(* CODESYS project TheWorld
   CompiledLibraryCompatibilityVersion: CODESYS V3.5 SP16 Patch 2

Project tree, tasks and I/O mapping:
  Device : CODESYS Control for Linux SL, CODESYS GmbH, order no. 2302000005, version 4.8.0.0
    application Application
      AC_FBs/
      AC_RMP/
      AC_Std/
      Alarm Configuration
      program BlinkingAlarm [CFC]
      program Calculus [ST]
      visualisation Chiller1Menu
      text list Chiller2Alarmgroup
      program Chiller_1 [ST]
      Chiller_func/
      text list Chiller_trendvalues
      function block ConvertDataArray_1 [ST]
      function block ConvertDataArray_2 [ST]
      function block ConvertDataArray_3 [ST]
      function block ConvertDataArray [ST]
      Enums/
    Ethernet : Ethernet, 3S - Smart Software Solutions GmbH, version 4.1.0.0 (disabled)
        settings: IPAddress = [172,16,0,11]; SubnetMask = [255,255,255,0]; GatewayAddress = [172,16,0,1]; MACAddress = [16#00,16#00,16#00,16#00,16#00,16#00]; NetworkInterfaceName = 'eno1'; NetworkInterfaceName = "eno1"; SaveCommunicationSettings = FALSE; IPAddress = [192,168,0,2]; SubnetMask = [255,255,255,0]; GatewayAddress = [0,0,0,0]
      Modbus_TCP_Master : Modbus TCP Master, 3S - Smart Software Solutions GmbH, version 4.2.0.0
          settings: AutoReconnect = TRUE
        Modbus_TCP_Slave_AC1 : Modbus TCP Slave, 3S - Smart Software Solutions GmbH, version 4.1.0.0
            settings: Unit-ID = 255; IPAddress = [192, 168, 0, 51]; Channel 0.Function Code = 3; Channel 0.Read Offset = 16#0000; Channel 0.Read Length = 124; Channel 0.Write Offset = 0; Channel 0.Write Length = 0; Channel 0.Cycle Time = 100; Channel 1.Function Code = 3; Channel 1.Read Offset = 16#007C; Channel 1.Read Length = 124; Channel 1.Write Offset = 0; Channel 1.Write Length = 0; Channel 1.Cycle Time = 100; Channel 2.Function Code = 3; Channel 2.Read Offset = 16#00F8; Channel 2.Read Length = 124; Channel 2.Write Offset = 0; Channel 2.Write Length = 0; Channel 2.Cycle Time = 100; Channel 3.Function Code = 16; Channel 3.Read Offset = 0; Channel 3.Read Length = 0; Channel 3.Write Offset = 16#011E; Channel 3.Write Length = 4; Channel 3.Cycle Time = 100
            input  Application.Chiller_1.modbus_var_1000 : ARRAY[0..123] OF WORD  // Channel 0
            input  Application.Chiller_1.modbus_var_1001 : ARRAY[0..123] OF WORD  // Channel 1
            input  Application.Chiller_1.modbus_var_1002 : ARRAY[0..123] OF WORD  // Channel 2
            output Application.Chiller_1.modbus_var_1002[286] : WORD  // Channel 3.Channel 3
            output Application.Chiller_1.modbus_var_1002[287] : WORD  // Channel 3.Channel 3
            output Application.Chiller_1.modbus_var_1002[288] : WORD  // Channel 3.Channel 3
            output Application.Chiller_1.modbus_var_1002[289] : WORD  // Channel 3.Channel 3
            unmapped channels: Channel 3
        Modbus_TCP_Slave_AC2 : Modbus TCP Slave, 3S - Smart Software Solutions GmbH, version 4.1.0.0
            settings: Unit-ID = 255; IPAddress = [192, 168, 0, 52]; Channel 0.Function Code = 3; Channel 0.Read Offset = 16#0000; Channel 0.Read Length = 124; Channel 0.Write Offset = 0; Channel 0.Write Length = 0; Channel 0.Cycle Time = 100; Channel 1.Function Code = 3; Channel 1.Read Offset = 16#007C; Channel 1.Read Length = 124; Channel 1.Write Offset = 0; Channel 1.Write Length = 0; Channel 1.Cycle Time = 100; Channel 2.Function Code = 3; Channel 2.Read Offset = 16#012C; Channel 2.Read Length = 100; Channel 2.Write Offset = 0; Channel 2.Write Length = 0; Channel 2.Cycle Time = 100
            input  Application.Chiller_2.modbus_var_1000 : ARRAY[0..123] OF WORD  // Channel 0
            input  Application.Chiller_2.modbus_var_1001 : ARRAY[0..123] OF WORD  // Channel 1
            input  Application.Chiller_2.modbus_var_1002 : ARRAY[0..99] OF WORD  // Channel 2
        Modbus_TCP_Slave_AC3 : Modbus TCP Slave, 3S - Smart Software Solutions GmbH, version 4.1.0.0
            settings: Unit-ID = 255; IPAddress = [192, 168, 0, 53]; Channel 0.Function Code = 3; Channel 0.Read Offset = 16#0000; Channel 0.Read Length = 124; Channel 0.Write Offset = 0; Channel 0.Write Length = 0; Channel 0.Cycle Time = 100; Channel 1.Function Code = 3; Channel 1.Read Offset = 16#007C; Channel 1.Read Length = 124; Channel 1.Write Offset = 0; Channel 1.Write Length = 0; Channel 1.Cycle Time = 100; Channel 2.Function Code = 3; Channel 2.Read Offset = 16#00F8; Channel 2.Read Length = 124; Channel 2.Write Offset = 0; Channel 2.Write Length = 0; Channel 2.Cycle Time = 100; Channel 3.Function Code = 16; Channel 3.Read Offset = 0; Channel 3.Read Length = 0; Channel 3.Write Offset = 16#011E; Channel 3.Write Length = 4; Channel 3.Cycle Time = 100
            input  Application.Chiller_3.modbus_var_1000 : ARRAY[0..123] OF WORD  // Channel 0
            input  Application.Chiller_3.modbus_var_1001 : ARRAY[0..123] OF WORD  // Channel 1
            input  Application.Chiller_3.modbus_var_1002 : ARRAY[0..123] OF WORD  // Channel 2
            output Application.Chiller_3.modbus_var_1002[286] : WORD  // Channel 3.Channel 3
            output Application.Chiller_3.modbus_var_1002[287] : WORD  // Channel 3.Channel 3
            output Application.Chiller_3.modbus_var_1002[288] : WORD  // Channel 3.Channel 3
            output Application.Chiller_3.modbus_var_1002[289] : WORD  // Channel 3.Channel 3
            unmapped channels: Channel 3
        Modbus_TCP_Slave_AC4 : Modbus TCP Slave, 3S - Smart Software Solutions GmbH, version 4.1.0.0
            settings: Unit-ID = 255; IPAddress = [192, 168, 0, 54]; Channel 0.Function Code = 3; Channel 0.Read Offset = 16#0000; Channel 0.Read Length = 124; Channel 0.Write Offset = 0; Channel 0.Write Length = 0; Channel 0.Cycle Time = 100; Channel 1.Function Code = 3; Channel 1.Read Offset = 16#007C; Channel 1.Read Length = 124; Channel 1.Write Offset = 0; Channel 1.Write Length = 0; Channel 1.Cycle Time = 100; Channel 2.Function Code = 3; Channel 2.Read Offset = 16#012C; Channel 2.Read Length = 100; Channel 2.Write Offset = 0; Channel 2.Write Length = 0; Channel 2.Cycle Time = 100
            input  Application.Chiller_4.modbus_var_1000 : ARRAY[0..123] OF WORD  // Channel 0
            input  Application.Chiller_4.modbus_var_1001 : ARRAY[0..123] OF WORD  // Channel 1
            input  Application.Chiller_4.modbus_var_1002 : ARRAY[0..99] OF WORD  // Channel 2
    Modbus_COM_1 : Modbus COM, 3S - Smart Software Solutions GmbH, version 3.5.16.0
        settings: DataBits = 8; StopBits = 1; ComPort = 1
      Modbus_Master_COM_Port_1 : Modbus Master, COM Port, 3S - Smart Software Solutions GmbH, version 4.2.0.0
          settings: Auto-restart communication = TRUE
        Modbus_Slave_COM_Port_AC1 : Modbus Slave, COM Port, 3S - Smart Software Solutions GmbH, version 3.5.16.0
            settings: SlaveAddress = 15; ResponseTimeout = 1000; UseExtendedFunctionCodes = TRUE; Channel 0.Function Code = 3; Channel 0.Read Offset = 16#0000; Channel 0.Read Length = 100; Channel 0.Write Offset = 0; Channel 0.Write Length = 0; Channel 0.Cycle Time = 100
            input  Application.Chiller_1.modbus_var_1000 : ARRAY[0..99] OF WORD  // Channel 0
        Modbus_Slave_COM_Port_AC2 : Modbus Slave, COM Port, 3S - Smart Software Solutions GmbH, version 3.5.16.0
            settings: SlaveAddress = 15; ResponseTimeout = 1000; UseExtendedFunctionCodes = TRUE; Channel 0.Function Code = 3; Channel 0.Read Offset = 16#0200; Channel 0.Read Length = 100; Channel 0.Write Offset = 0; Channel 0.Write Length = 0; Channel 0.Cycle Time = 100
            input  Application.Chiller_2.modbus_var_1000 : ARRAY[0..99] OF WORD  // Channel 0
        Modbus_Slave_COM_Port_AC3 : Modbus Slave, COM Port, 3S - Smart Software Solutions GmbH, version 3.5.16.0
            settings: SlaveAddress = 16; ResponseTimeout = 1000; UseExtendedFunctionCodes = TRUE; Channel 0.Function Code = 3; Channel 0.Read Offset = 16#0400; Channel 0.Read Length = 100; Channel 0.Write Offset = 0; Channel 0.Write Length = 0; Channel 0.Cycle Time = 100
            input  Application.Chiller_3.modbus_var_1000 : ARRAY[0..99] OF WORD  // Channel 0
        Modbus_Slave_COM_Port_AC4 : Modbus Slave, COM Port, 3S - Smart Software Solutions GmbH, version 3.5.16.0
            settings: SlaveAddress = 16; ResponseTimeout = 1000; UseExtendedFunctionCodes = TRUE; Channel 0.Function Code = 3; Channel 0.Read Offset = 16#0600; Channel 0.Read Length = 100; Channel 0.Write Offset = 0; Channel 0.Write Length = 0; Channel 0.Cycle Time = 100
            input  Application.Chiller_4.modbus_var_1000 : ARRAY[0..99] OF WORD  // Channel 0
        Modbus_Slave_COM_Port_AC5 : Modbus Slave, COM Port, 3S - Smart Software Solutions GmbH, version 3.5.16.0
            settings: SlaveAddress = 16; ResponseTimeout = 1000; UseExtendedFunctionCodes = TRUE; Channel 0.Function Code = 3; Channel 0.Read Offset = 16#0800; Channel 0.Read Length = 100; Channel 0.Write Offset = 0; Channel 0.Write Length = 0; Channel 0.Cycle Time = 100
            input  Application.Chiller_5.modbus_var_1000 : ARRAY[0..99] OF WORD  // Channel 0
        Modbus_Slave_COM_Port_AC6 : Modbus Slave, COM Port, 3S - Smart Software Solutions GmbH, version 3.5.16.0
            settings: SlaveAddress = 16; ResponseTimeout = 1000; UseExtendedFunctionCodes = TRUE; Channel 0.Function Code = 3; Channel 0.Read Offset = 16#0C00; Channel 0.Read Length = 100; Channel 0.Write Offset = 0; Channel 0.Write Length = 0; Channel 0.Cycle Time = 100
            input  Application.Chiller_6.modbus_var_1000 : ARRAY[0..99] OF WORD  // Channel 0
        Modbus_Slave_COM_Seq : Modbus Slave, COM Port, 3S - Smart Software Solutions GmbH, version 3.5.16.0
            settings: SlaveAddress = 16; ResponseTimeout = 1000; UseExtendedFunctionCodes = TRUE; Channel 0.Function Code = 3; Channel 0.Read Offset = 16#0A00; Channel 0.Read Length = 108; Channel 0.Write Offset = 0; Channel 0.Write Length = 0; Channel 0.Cycle Time = 100; Channel 1.Function Code = 3; Channel 1.Read Offset = 16#0A7C; Channel 1.Read Length = 83; Channel 1.Write Offset = 0; Channel 1.Write Length = 0; Channel 1.Cycle Time = 100
            input  Application.Sequence.modbus_var_1000 : ARRAY[0..107] OF WORD  // Channel 0
            input  Application.Sequence.modbus_var_add : ARRAY[0..82] OF WORD  // Channel 1
    Modbus_COM_1 : Modbus COM, 3S - Smart Software Solutions GmbH, version 4.1.0.0
      Modbus_Master_COM_Port_1 : Modbus Master, COM Port, 3S - Smart Software Solutions GmbH, version 4.3.0.0
          settings: Transmission = 'RTU'; ResponseTimeout = 1000; TimeBetweenFrames = 10; Auto-restart communication = TRUE
        Modbus_Slave_AC1 : Modbus Slave, COM Port, 3S - Smart Software Solutions GmbH, version 4.1.0.0
            settings: SlaveAddress = 15; ResponseTimeout = 1000; UseExtendedFunctionCodes = TRUE; Channel 0.Function Code = 3; Channel 0.Read Offset = 16#0000; Channel 0.Read Length = 60; Channel 0.Write Offset = 0; Channel 0.Write Length = 0; Channel 0.Cycle Time = 100
            input  Application.Chiller_1.modbus_var_1000 : ARRAY[0..59] OF WORD  // Channel 0
        Modbus_Slave_AC2 : Modbus Slave, COM Port, 3S - Smart Software Solutions GmbH, version 4.1.0.0
            settings: SlaveAddress = 15; ResponseTimeout = 1000; UseExtendedFunctionCodes = TRUE; Channel 0.Function Code = 3; Channel 0.Read Offset = 16#0200; Channel 0.Read Length = 60; Channel 0.Write Offset = 0; Channel 0.Write Length = 0; Channel 0.Cycle Time = 100
            input  Application.Chiller_2.modbus_var_1000 : ARRAY[0..59] OF WORD  // Channel 0
        Modbus_Slave_AC3 : Modbus Slave, COM Port, 3S - Smart Software Solutions GmbH, version 4.1.0.0
            settings: SlaveAddress = 15; ResponseTimeout = 1000; UseExtendedFunctionCodes = TRUE; Channel 0.Function Code = 3; Channel 0.Read Offset = 16#0400; Channel 0.Read Length = 60; Channel 0.Write Offset = 0; Channel 0.Write Length = 0; Channel 0.Cycle Time = 100
            input  Application.Chiller_3.modbus_var_1000 : ARRAY[0..59] OF WORD  // Channel 0
    SoftMotion General Axis Pool
  libraries: CmpBitmapPool, 3.5.17.0 (System); AC_DataLog, 3.5.16.0 (3S - Smart Software Solutions GmbH)
  5ce3da45-db07-42e7-a21c-a00fff4ed8f6|C:\Users\Codesys\Desktop\FlowDiagram_Edited.PNG
  5ce3da45-db07-42e7-a21c-a00fff4ed8f6|C:\Users\Codesys\Desktop\FlowDiagram_Edited.PNG
  5ce3da45-db07-42e7-a21c-a00fff4ed8f6|C:\Users\Codesys\Desktop\Images\Assets från KT_PC\VSD\VSD.jpg
  5ce3da45-db07-42e7-a21c-a00fff4ed8f6|C:\Users\Codesys\Desktop\Images\Assets från KT_PC\VSD\VSD.jpg
  5ce3da45-db07-42e7-a21c-a00fff4ed8f6|C:\Users\Codesys\Desktop\Images\Div bilder\Arrow gray left.png
  5ce3da45-db07-42e7-a21c-a00fff4ed8f6|C:\Users\Codesys\Desktop\Images\Div bilder\Arrow gray left.png
  5ce3da45-db07-42e7-a21c-a00fff4ed8f6|C:\Users\Codesys\Desktop\Images\Div bilder\Arrow green down.png
  5ce3da45-db07-42e7-a21c-a00fff4ed8f6|C:\Users\Codesys\Desktop\Images\Div bilder\Arrow green down.png
  5ce3da45-db07-42e7-a21c-a00fff4ed8f6|C:\Users\Codesys\Desktop\Images\Div bilder\Arrow green up.png
  5ce3da45-db07-42e7-a21c-a00fff4ed8f6|C:\Users\Codesys\Desktop\Images\Div bilder\Arrow green up.png
  5ce3da45-db07-42e7-a21c-a00fff4ed8f6|C:\Users\Codesys\Desktop\Images\Div bilder\Arrow lightblue left.png
  5ce3da45-db07-42e7-a21c-a00fff4ed8f6|C:\Users\Codesys\Desktop\Images\Div bilder\Arrow lightblue left.png
  5ce3da45-db07-42e7-a21c-a00fff4ed8f6|C:\Users\Codesys\Desktop\Images\Div bilder\Arrow red down.png
  5ce3da45-db07-42e7-a21c-a00fff4ed8f6|C:\Users\Codesys\Desktop\Images\Div bilder\Arrow red down.png
  5ce3da45-db07-42e7-a21c-a00fff4ed8f6|C:\Users\Codesys\Desktop\Images\Div bilder\Arrow red left.png
  5ce3da45-db07-42e7-a21c-a00fff4ed8f6|C:\Users\Codesys\Desktop\Images\Div bilder\Arrow red left.png
  5ce3da45-db07-42e7-a21c-a00fff4ed8f6|C:\Users\Codesys\Desktop\Images\Invisible.png
  5ce3da45-db07-42e7-a21c-a00fff4ed8f6|C:\Users\Codesys\Desktop\Images\Invisible.png
  5ce3da45-db07-42e7-a21c-a00fff4ed8f6|C:\Users\Codesys\Desktop\Images\LEDS\ALARM.png
  5ce3da45-db07-42e7-a21c-a00fff4ed8f6|C:\Users\Codesys\Desktop\Images\LEDS\ALARM.png
  5ce3da45-db07-42e7-a21c-a00fff4ed8f6|C:\Users\Codesys\Desktop\Images\LEDS\Led_SQ_Green1_On_Medium.png
  5ce3da45-db07-42e7-a21c-a00fff4ed8f6|C:\Users\Codesys\Desktop\Images\LEDS\Led_SQ_Green1_On_Medium.png
  5ce3da45-db07-42e7-a21c-a00fff4ed8f6|C:\Users\Codesys\Desktop\Images\LEDS\Led_SQ_Grey_Off_Medium.png
  5ce3da45-db07-42e7-a21c-a00fff4ed8f6|C:\Users\Codesys\Desktop\Images\LEDS\Led_SQ_Grey_Off_Medium.png
  5ce3da45-db07-42e7-a21c-a00fff4ed8f6|C:\Users\Codesys\Desktop\Images\LEDS\TRIP.png
  5ce3da45-db07-42e7-a21c-a00fff4ed8f6|C:\Users\Codesys\Desktop\Images\LEDS\TRIP.png
  5ce3da45-db07-42e7-a21c-a00fff4ed8f6|C:\Users\Codesys\Desktop\Images\Logo-Aida.png
  5ce3da45-db07-42e7-a21c-a00fff4ed8f6|C:\Users\Codesys\Desktop\Images\Logo-Aida.png
  5ce3da45-db07-42e7-a21c-a00fff4ed8f6|C:\Users\Codesys\Desktop\Images\Logo-Costa.png
  5ce3da45-db07-42e7-a21c-a00fff4ed8f6|C:\Users\Codesys\Desktop\Images\Logo-Costa.png
  5ce3da45-db07-42e7-a21c-a00fff4ed8f6|C:\Users\Codesys\Desktop\Images\Logo-HAL.png
  5ce3da45-db07-42e7-a21c-a00fff4ed8f6|C:\Users\Codesys\Desktop\Images\Logo-HAL.png
  5ce3da45-db07-42e7-a21c-a00fff4ed8f6|C:\Users\Codesys\Desktop\Images\Logo-ncl.png
  5ce3da45-db07-42e7-a21c-a00fff4ed8f6|C:\Users\Codesys\Desktop\Images\Logo-ncl.png
  5ce3da45-db07-42e7-a21c-a00fff4ed8f6|C:\Users\Codesys\Desktop\Images\Logo-Princess.png
  5ce3da45-db07-42e7-a21c-a00fff4ed8f6|C:\Users\Codesys\Desktop\Images\Logo-Princess.png
  5ce3da45-db07-42e7-a21c-a00fff4ed8f6|C:\Users\Codesys\Desktop\Images\Logo-TUI.png
  5ce3da45-db07-42e7-a21c-a00fff4ed8f6|C:\Users\Codesys\Desktop\Images\Logo-TUI.png
  5ce3da45-db07-42e7-a21c-a00fff4ed8f6|C:\Users\Codesys\Desktop\Images\Menu\AlarmMenu.png
  5ce3da45-db07-42e7-a21c-a00fff4ed8f6|C:\Users\Codesys\Desktop\Images\Menu\AlarmMenu.png
  5ce3da45-db07-42e7-a21c-a00fff4ed8f6|C:\Users\Codesys\Desktop\Images\Menu\EventMenu.png
  5ce3da45-db07-42e7-a21c-a00fff4ed8f6|C:\Users\Codesys\Desktop\Images\Pipes\PipeGreen_1_Horizontal.png
  5ce3da45-db07-42e7-a21c-a00fff4ed8f6|C:\Users\Codesys\Desktop\Images\Pipes\PipeGreen_1_Horizontal.png
  5ce3da45-db07-42e7-a21c-a00fff4ed8f6|C:\Users\Codesys\Desktop\Images\Pipes\PipeGreen_1_LD.png
  5ce3da45-db07-42e7-a21c-a00fff4ed8f6|C:\Users\Codesys\Desktop\Images\Pipes\PipeGreen_1_LD.png
  5ce3da45-db07-42e7-a21c-a00fff4ed8f6|C:\Users\Codesys\Desktop\Images\Pipes\PipeGreen_2_LU.png
  5ce3da45-db07-42e7-a21c-a00fff4ed8f6|C:\Users\Codesys\Desktop\Images\Pipes\PipeGreen_2_LU.png
  5ce3da45-db07-42e7-a21c-a00fff4ed8f6|C:\Users\Codesys\Desktop\Images\Pipes\PipeGreen_3way_2.png
  5ce3da45-db07-42e7-a21c-a00fff4ed8f6|C:\Users\Codesys\Desktop\Images\Pipes\PipeGreen_3way_2.png
  5ce3da45-db07-42e7-a21c-a00fff4ed8f6|C:\Users\Codesys\Desktop\Images\Pipes\PipeGreen_3way.png
  5ce3da45-db07-42e7-a21c-a00fff4ed8f6|C:\Users\Codesys\Desktop\Images\Pipes\PipeGreen_3way.png
  5ce3da45-db07-42e7-a21c-a00fff4ed8f6|C:\Users\Codesys\Desktop\Images\Pipes\PipeGrey_1S_Horizontal.png
  5ce3da45-db07-42e7-a21c-a00fff4ed8f6|C:\Users\Codesys\Desktop\Images\Pipes\PipeGrey_1S_Horizontal.png
  5ce3da45-db07-42e7-a21c-a00fff4ed8f6|C:\Users\Codesys\Desktop\Images\Pipes\PipeGrey_2_LD.png
  5ce3da45-db07-42e7-a21c-a00fff4ed8f6|C:\Users\Codesys\Desktop\Images\Pipes\PipeGrey_2_LD.png
  5ce3da45-db07-42e7-a21c-a00fff4ed8f6|C:\Users\Codesys\Desktop\Images\Pipes\PipeGrey_3_LU.png
  5ce3da45-db07-42e7-a21c-a00fff4ed8f6|C:\Users\Codesys\Desktop\Images\Pipes\PipeGrey_3_LU.png
  5ce3da45-db07-42e7-a21c-a00fff4ed8f6|C:\Users\Codesys\Desktop\Images\Pipes\PipeLightBlue_1_Horizontal.png
  5ce3da45-db07-42e7-a21c-a00fff4ed8f6|C:\Users\Codesys\Desktop\Images\Pipes\PipeLightBlue_1_Horizontal.png
  5ce3da45-db07-42e7-a21c-a00fff4ed8f6|C:\Users\Codesys\Desktop\Images\Pipes\PipeLightBlue_1_LD.png
  5ce3da45-db07-42e7-a21c-a00fff4ed8f6|C:\Users\Codesys\Desktop\Images\Pipes\PipeLightBlue_1_LD.png
  5ce3da45-db07-42e7-a21c-a00fff4ed8f6|C:\Users\Codesys\Desktop\Images\Pipes\PipeLightBlue_1_Vertical.png
  5ce3da45-db07-42e7-a21c-a00fff4ed8f6|C:\Users\Codesys\Desktop\Images\Pipes\PipeLightBlue_1_Vertical.png
  5ce3da45-db07-42e7-a21c-a00fff4ed8f6|C:\Users\Codesys\Desktop\Images\Pipes\PipeLightBlue_2_LU.png
  5ce3da45-db07-42e7-a21c-a00fff4ed8f6|C:\Users\Codesys\Desktop\Images\Pipes\PipeLightBlue_2_LU.png
  5ce3da45-db07-42e7-a21c-a00fff4ed8f6|C:\Users\Codesys\Desktop\Images\Pipes\PipeLightBlue_3_RD.png
  5ce3da45-db07-42e7-a21c-a00fff4ed8f6|C:\Users\Codesys\Desktop\Images\Pipes\PipeLightBlue_3_RD.png
  5ce3da45-db07-42e7-a21c-a00fff4ed8f6|C:\Users\Codesys\Desktop\Images\Pipes\PipeLightBlue_3_RU.png
  5ce3da45-db07-42e7-a21c-a00fff4ed8f6|C:\Users\Codesys\Desktop\Images\Pipes\PipeLightBlue_3_RU.png
  5ce3da45-db07-42e7-a21c-a00fff4ed8f6|C:\Users\Codesys\Desktop\Images\Pipes\PipeRed_1_LD.png
  5ce3da45-db07-42e7-a21c-a00fff4ed8f6|C:\Users\Codesys\Desktop\Images\Pipes\PipeRed_1_LD.png
  5ce3da45-db07-42e7-a21c-a00fff4ed8f6|C:\Users\Codesys\Desktop\Images\Pipes\PipeRed_1_RD.png
  5ce3da45-db07-42e7-a21c-a00fff4ed8f6|C:\Users\Codesys\Desktop\Images\Pipes\PipeRed_1_RD.png
  5ce3da45-db07-42e7-a21c-a00fff4ed8f6|C:\Users\Codesys\Desktop\Images\Pipes\PipeRed_2_Horizontal.png
  5ce3da45-db07-42e7-a21c-a00fff4ed8f6|C:\Users\Codesys\Desktop\Images\Pipes\PipeRed_2_Horizontal.png
  5ce3da45-db07-42e7-a21c-a00fff4ed8f6|C:\Users\Codesys\Desktop\Images\Pipes\PipeRed_2_LU.png
  5ce3da45-db07-42e7-a21c-a00fff4ed8f6|C:\Users\Codesys\Desktop\Images\Pipes\PipeRed_2_LU.png
  5ce3da45-db07-42e7-a21c-a00fff4ed8f6|C:\Users\Codesys\Desktop\Images\Pipes\PipeRed_2_RU.png
  5ce3da45-db07-42e7-a21c-a00fff4ed8f6|C:\Users\Codesys\Desktop\Images\Pipes\PipeRed_2_RU.png
  5ce3da45-db07-42e7-a21c-a00fff4ed8f6|C:\Users\Codesys\Desktop\Images\Pumps\Pump_Large_3.png
  5ce3da45-db07-42e7-a21c-a00fff4ed8f6|C:\Users\Codesys\Desktop\Images\Pumps\Pump_Large_3.png
  5ce3da45-db07-42e7-a21c-a00fff4ed8f6|C:\Users\Codesys\Desktop\Images\Scales\BarScale3.png
  5ce3da45-db07-42e7-a21c-a00fff4ed8f6|C:\Users\Codesys\Desktop\Images\Scales\BarScale3.png
  5ce3da45-db07-42e7-a21c-a00fff4ed8f6|C:\Users\Codesys\Desktop\Images\Scales\BarScale4.png
  5ce3da45-db07-42e7-a21c-a00fff4ed8f6|C:\Users\Codesys\Desktop\Images\Scales\BarScale4.png
  5ce3da45-db07-42e7-a21c-a00fff4ed8f6|C:\Users\Codesys\Desktop\Images\Ships\Norwegian Joy.jpg
  5ce3da45-db07-42e7-a21c-a00fff4ed8f6|C:\Users\Codesys\Desktop\Images\Transparants\CapBarTranparant.png
  5ce3da45-db07-42e7-a21c-a00fff4ed8f6|C:\Users\Codesys\Desktop\Images\Transparants\CapBarTranparant.png
  5ce3da45-db07-42e7-a21c-a00fff4ed8f6|C:\Users\Codesys\Desktop\Images\Valves\Valve_2.png
  5ce3da45-db07-42e7-a21c-a00fff4ed8f6|C:\Users\Codesys\Desktop\Images\Valves\Valve_2.png
  5ce3da45-db07-42e7-a21c-a00fff4ed8f6|C:\Users\Codesys\Desktop\Images\Valves\Valve_3.png
  5ce3da45-db07-42e7-a21c-a00fff4ed8f6|C:\Users\Codesys\Desktop\Images\Valves\Valve_3.png
  5ce3da45-db07-42e7-a21c-a00fff4ed8f6|C:\Users\Codesys\Desktop\Images\Valves\Valve_4.png
  5ce3da45-db07-42e7-a21c-a00fff4ed8f6|C:\Users\Codesys\Desktop\Images\Valves\Valve_4.png
  5ce3da45-db07-42e7-a21c-a00fff4ed8f6|C:\Users\Codesys\Desktop\MenuAlarm.png
  5ce3da45-db07-42e7-a21c-a00fff4ed8f6|C:\Users\Codesys\Desktop\MenuAlarm.png
  5ce3da45-db07-42e7-a21c-a00fff4ed8f6|C:\Users\Codesys\Desktop\MenuEvents.png
  5ce3da45-db07-42e7-a21c-a00fff4ed8f6|C:\Users\Codesys\Desktop\MenuEvents.png
  5ce3da45-db07-42e7-a21c-a00fff4ed8f6|C:\Users\Codesys\Desktop\MenuHome.png
  5ce3da45-db07-42e7-a21c-a00fff4ed8f6|C:\Users\Codesys\Desktop\MenuHome.png
  5ce3da45-db07-42e7-a21c-a00fff4ed8f6|C:\Users\Codesys\Desktop\MenuLogout.png
  5ce3da45-db07-42e7-a21c-a00fff4ed8f6|C:\Users\Codesys\Desktop\MenuLogout.png
  5ce3da45-db07-42e7-a21c-a00fff4ed8f6|C:\Users\Codesys\Desktop\MenuSchematics.png
  5ce3da45-db07-42e7-a21c-a00fff4ed8f6|C:\Users\Codesys\Desktop\MenuSchematics.png
  5ce3da45-db07-42e7-a21c-a00fff4ed8f6|C:\Users\Codesys\Desktop\MenuSettings.png
  5ce3da45-db07-42e7-a21c-a00fff4ed8f6|C:\Users\Codesys\Desktop\MenuSettings.png
  5ce3da45-db07-42e7-a21c-a00fff4ed8f6|C:\Users\Codesys\Desktop\ncl_breakaway.jpg
  5ce3da45-db07-42e7-a21c-a00fff4ed8f6|C:\Users\Codesys\Desktop\VSD_Edited.png
  5ce3da45-db07-42e7-a21c-a00fff4ed8f6|C:\Users\Codesys\Desktop\white.PNG
  5ce3da45-db07-42e7-a21c-a00fff4ed8f6|C:\Users\Codesys\Desktop\white.PNG
  5ce3da45-db07-42e7-a21c-a00fff4ed8f6|C:\Users\Codesys\Documents\logo\1200px-Johnson_Controls.svg.png
  5ce3da45-db07-42e7-a21c-a00fff4ed8f6|C:\Users\Codesys\Documents\logo\1200px-Johnson_Controls.svg.png
  5ce3da45-db07-42e7-a21c-a00fff4ed8f6|C:\Users\Codesys\Documents\logo\JCI_Full Color_Transparent Background.png
  5ce3da45-db07-42e7-a21c-a00fff4ed8f6|C:\Users\Codesys\Documents\logo\JCI_Full Color_Transparent Background.png
  5ce3da45-db07-42e7-a21c-a00fff4ed8f6|C:\Users\Codesys\Pictures\ConquestVSChiller1.jpg
  5ce3da45-db07-42e7-a21c-a00fff4ed8f6|C:\Users\Codesys\Pictures\ConquestVSChiller1.jpg
  5ce3da45-db07-42e7-a21c-a00fff4ed8f6|C:\Users\Codesys\Pictures\ConquestVSChiller.jpg
  5ce3da45-db07-42e7-a21c-a00fff4ed8f6|C:\Users\Codesys\Pictures\Grafic_oldradar\2016_update\Images\Chiller\Compressor.png
  5ce3da45-db07-42e7-a21c-a00fff4ed8f6|C:\Users\Codesys\Pictures\Grafic_oldradar\2016_update\Images\Chiller\Compressor.png
  5ce3da45-db07-42e7-a21c-a00fff4ed8f6|C:\Users\Codesys\Pictures\Grafic_oldradar\2016_update\Images\Chiller\Condenser.png
  5ce3da45-db07-42e7-a21c-a00fff4ed8f6|C:\Users\Codesys\Pictures\Grafic_oldradar\2016_update\Images\Chiller\Condenser.png
  5ce3da45-db07-42e7-a21c-a00fff4ed8f6|C:\Users\Codesys\Pictures\Grafic_oldradar\2016_update\Images\Chiller\Evaporator3.png
  5ce3da45-db07-42e7-a21c-a00fff4ed8f6|C:\Users\Codesys\Pictures\Grafic_oldradar\2016_update\Images\Chiller\Evaporator.png
  5ce3da45-db07-42e7-a21c-a00fff4ed8f6|C:\Users\Codesys\Pictures\Grafic_oldradar\2016_update\Images\Chiller\Evaporator.png
  5ce3da45-db07-42e7-a21c-a00fff4ed8f6|C:\Users\Codesys\Pictures\Grafic_oldradar\2016_update\Images\Pipes\PipeGrey_1_LU.png
  5ce3da45-db07-42e7-a21c-a00fff4ed8f6|C:\Users\Codesys\Pictures\Grafic_oldradar\2016_update\Images\Pipes\PipeGrey_1_RD.png
  5ce3da45-db07-42e7-a21c-a00fff4ed8f6|C:\Users\Codesys\Pictures\Grafic_oldradar\2016_update\Images\Pipes\PipeGrey_1S_Horizontal.png
  5ce3da45-db07-42e7-a21c-a00fff4ed8f6|C:\Users\Codesys\Pictures\islandP.jpg
  5ce3da45-db07-42e7-a21c-a00fff4ed8f6|C:\Users\Codesys\Pictures\Sapphire_Princess_sing.jpg
  5ce3da45-db07-42e7-a21c-a00fff4ed8f6|C:\Users\Technician\Desktop\NCL_Bliss.jpg
  5ce3da45-db07-42e7-a21c-a00fff4ed8f6|C:\Users\Technician\Documents\Codesys\Export\the-world-2.jpg
  5ce3da45-db07-42e7-a21c-a00fff4ed8f6|C:\Users\Technician\Documents\Codesys\Export\TheWorldLogo.png
  5ce3da45-db07-42e7-a21c-a00fff4ed8f6|C:\Users\Technician\Pictures\NCL Encore 4 (bäst).jpg
  5ce3da45-db07-42e7-a21c-a00fff4ed8f6|C:\Users\User\Desktop\FlowDiagram_Edited.PNG
  5ce3da45-db07-42e7-a21c-a00fff4ed8f6|E:\Images\Images\Chiller\ACChiller3D.png
  5ce3da45-db07-42e7-a21c-a00fff4ed8f6|E:\Images\Images\Chiller\ACChiller3D.png
  AC_GENERATOR_DATA
  DataLogManager
    Channels for DataLog (DataLogChannels)
      DataLogChannel_1
        A storage module. (DataLogStorage)
        DataLogStorage1_CSV
      DataLogChannel_2
        A storage module. (DataLogStorage)
        DataLogStorage_CSV2
      DataLogChannel_3
        A storage module. (DataLogStorage)
        DataLogStorage_CSV3
      DataLogChannel_4
        A storage module. (DataLogStorage)
        DataLogStorage_CSV4
      DataLogChannel
        A storage module. (DataLogStorage)
        DataLogStorage_CSV
  text list GlobalTextList
  PersistenceManager
    Channels (pChannels)
      PersistenceChannel
  text list System
*)

// Device/Application/BlinkingAlarm
PROGRAM BlinkingAlarm
VAR
	TimeOn: TIME:= T#1S;
	TimeOff: TIME:= T#1S;
	Alarm: BOOL;
	TurnOn: BOOL;
		
	Blink_0: BLINK;
	
END_VAR
VAR // added by the converter: edge detectors and wires of the graphical bodies
    _w1, _w2 : BOOL;
END_VAR

TurnOn := _w1;
_w1 := not.Sequence.Alarm_sequence OR not.Chiller_1.Unit_alarm OR not.Chiller_1.Unit_trip OR not.Chiller_2.Unit_alarm OR not.Chiller_2.Unit_trip OR not.Chiller_3.Unit_alarm OR not.Chiller_3.Unit_trip OR not.Chiller_4.Unit_alarm OR not.Chiller_4.Unit_trip;
_w2 := TurnOn AND Blink_0.OUT;
Blink_0(ENABLE := TurnOn, TIMELOW := TimeOff, TIMEHIGH := TimeOn); // BLINK
Alarm := _w2;

END_PROGRAM

// Device/Application/Chiller_1
PROGRAM Chiller_1
VAR

timer2 : standard.ton ;
{attribute 'ac_datalog_set_default_group' := 'DataLogChannel'}
instStruct : LogStruct;


modbus_var : ARRAY[0..100] OF INT;
modbus_var_1000 : ARRAY[0..123] OF WORD;
modbus_var_1001 : ARRAY[124..247] OF WORD;
modbus_var_1002 : ARRAY[248..371] OF WORD;
{attribute 'ac_datalog_hysteresis' := '0.2'}
{attribute 'ac_datalog' := 'DatalogChannel'}
Temp_chilled_medium_out : REAL;
{attribute 'ac_datalog_hysteresis' := '0.2'}
{attribute 'ac_datalog' := 'DatalogChannel'}
Temp_chilled_medium_in : REAL;
{attribute 'ac_datalog_hysteresis' := '0.2'}
{attribute 'ac_datalog' := 'DatalogChannel'}
Temp_water_inlet_cond : REAL;
{attribute 'ac_datalog_hysteresis' := '0.2'}
{attribute 'ac_datalog' := 'DatalogChannel'}
Press_suction_compr : REAL;
{attribute 'ac_datalog_hysteresis' := '0.5'}
{attribute 'ac_datalog' := 'DatalogChannel'}
Press_discharge_compr : REAL;
{attribute 'ac_datalog_hysteresis' := '0.5'}
{attribute 'ac_datalog' := 'DatalogChannel'}
Press_oil_receiver : REAL;
{attribute 'ac_datalog_hysteresis' := '0.5'}
{attribute 'ac_datalog' := 'DatalogChannel'}
Press_oil_compr : REAL;
{attribute 'ac_datalog_hysteresis' := '0.4'}
{attribute 'ac_datalog' := 'DatalogChannel'}
Temp_discharge : REAL;
{attribute 'ac_datalog_hysteresis' := '0.5'}
{attribute 'ac_datalog' := 'DatalogChannel'}
Oil_temp_receiver : REAL;
{attribute 'ac_datalog_hysteresis' := '0.5'}
{attribute 'ac_datalog' := 'DatalogChannel'}
Max_motor_temp : REAL;
{attribute 'ac_datalog_hysteresis' := '0.2'}
{attribute 'ac_datalog' := 'DatalogChannel'}
Temp_motor_bearing_DE : REAL;
{attribute 'ac_datalog_hysteresis' := '0.2'}
{attribute 'ac_datalog' := 'DatalogChannel'}
Temp_motor_bearing_NDE : REAL;
{attribute 'ac_datalog_hysteresis' := '4'}
{attribute 'ac_datalog' := 'DatalogChannel'}
Motor_current : REAL;
{attribute 'ac_datalog_hysteresis' := '50'}
{attribute 'ac_datalog' := 'DatalogChannel'}
Running_hours_comp_unscaled : WORD;
{attribute 'ac_datalog_hysteresis' := '50'}
{attribute 'ac_datalog' := 'DatalogChannel'}
Running_hours_oil_pump_unscaled : WORD;
{attribute 'ac_datalog' := 'DatalogChannel'}
Anti_recycle_time : REAL;
{attribute 'ac_datalog_hysteresis' := '2'}
{attribute 'ac_datalog' := 'DatalogChannel'}
Feedback_compressor : REAL;
{attribute 'ac_datalog_hysteresis' := '0.2'}
{attribute 'ac_datalog' := 'DatalogChannel'}
Oil_diff_pressure : REAL;
{attribute 'ac_datalog_hysteresis' := '0.3'}
{attribute 'ac_datalog' := 'DatalogChannel'}
Suction_saturated_temp : REAL;
{attribute 'ac_datalog_hysteresis' := '0.2'}
{attribute 'ac_datalog' := 'DatalogChannel'}
Discharge_saturated_temp : REAL;
{attribute 'ac_datalog_hysteresis' := '0.2'}
{attribute 'ac_datalog' := 'DatalogChannel'}
Temp_water_outlet_cond : REAL;
{attribute 'ac_datalog_hysteresis' := '0.2'}
{attribute 'ac_datalog' := 'DatalogChannel'}
Temp_motor_wind_R : REAL;
{attribute 'ac_datalog_hysteresis' := '0.2'}
{attribute 'ac_datalog' := 'DatalogChannel'}
Temp_motor_wind_S : REAL;
{attribute 'ac_datalog_hysteresis' := '0.2'}
{attribute 'ac_datalog' := 'DatalogChannel'}
Temp_motor_wind_T : REAL;
{attribute 'ac_datalog_hysteresis' := '0.2'}
{attribute 'ac_datalog' := 'DatalogChannel'}
Temp_motor_air : REAL;
{attribute 'ac_datalog_hysteresis' := '0.04'}
{attribute 'ac_datalog' := 'DatalogChannel'}
dP_CW : REAL;
{attribute 'ac_datalog_hysteresis' := '0.04'}
{attribute 'ac_datalog' := 'DatalogChannel'}
dP_SW : REAL;
{attribute 'ac_datalog_hysteresis' := '4'}
{attribute 'ac_datalog' := 'DatalogChannel'}
Chiller_capacity : REAL;
{attribute 'ac_datalog_hysteresis' := '2'}
{attribute 'ac_datalog' := 'DatalogChannel'}
Temp_oil_inlet_compr : REAL;
Spare : REAL;
{attribute 'ac_datalog_hysteresis' := '2'}
{attribute 'ac_datalog' := 'DatalogChannel'}
SP_CW_controller : REAL;
{attribute 'ac_datalog_hysteresis' := '2'}
{attribute 'ac_datalog' := 'DatalogChannel'}
Setpoint_oil_pump : REAL;
{attribute 'ac_datalog_hysteresis' := '0.02'}
{attribute 'ac_datalog' := 'DatalogChannel'}
Thrust_bearing_position : REAL;
{attribute 'ac_datalog_hysteresis' := '50'}
{attribute 'ac_datalog' := 'DatalogChannel'}
Oil_pump_running_hours : REAL;
{attribute 'ac_datalog_hysteresis' := '5'}
{attribute 'ac_datalog' := 'DatalogChannel'}
Liquid_level_condenser : REAL;
{attribute 'ac_datalog_hysteresis' := '0.05'}
{attribute 'ac_datalog' := 'DatalogChannel'}
Oil_Filter_Drop : REAL; 
{attribute 'ac_datalog_hysteresis' := '2'}
{attribute 'ac_datalog' := 'DatalogChannel'}
Proximitor_thrust_pos : REAL;
{attribute 'ac_datalog_hysteresis' := '0.4'}
{attribute 'ac_datalog' := 'DatalogChannel'}
Press_chilled_medium_in : REAL;
{attribute 'ac_datalog_hysteresis' := '0.2'}
{attribute 'ac_datalog' := 'DatalogChannel'}
Press_water_cond_out : REAL;
{attribute 'ac_datalog_hysteresis' := '0.02'}
{attribute 'ac_datalog' := 'DatalogChannel'}
Feedback_sea_water_valve : REAL;
{attribute 'ac_datalog_hysteresis' := '1'}
{attribute 'ac_datalog' := 'DatalogChannel'}
Oil_pressure_before_filter : REAL;
{attribute 'ac_datalog_hysteresis' := '0.2'}
{attribute 'ac_datalog' := 'DatalogChannel'}
Trafo_winding_temp : REAL;
{attribute 'ac_datalog_hysteresis' := '1'}
{attribute 'ac_datalog' := 'DatalogChannel'}
Feedback_VGD : REAL;
{attribute 'ac_datalog_hysteresis' := '4'}
{attribute 'ac_datalog' := 'DatalogChannel'}
Feedback_liquid_valve : REAL;
{attribute 'ac_datalog_hysteresis' := '3'}
{attribute 'ac_datalog' := 'DatalogChannel'}
Feedback_HGV : REAL;
{attribute 'ac_datalog_hysteresis' := '2'}
{attribute 'ac_datalog' := 'DatalogChannel'}
Discharge_superheat : REAL;
{attribute 'ac_datalog_hysteresis' := '0.6'}
{attribute 'ac_datalog' := 'DatalogChannel'}
Frequency_oil_pump : REAL;
{attribute 'ac_datalog_hysteresis' := '3'}
{attribute 'ac_datalog' := 'DatalogChannel'}
Hot_gas_valve_output : REAL;
{attribute 'ac_datalog_hysteresis' := '2'}
{attribute 'ac_datalog' := 'DatalogChannel'}
Control_signal_unit_d : REAL;
{attribute 'ac_datalog_hysteresis' := '2'}
{attribute 'ac_datalog' := 'DatalogChannel'}
Stall_detector : REAL;
{attribute 'ac_datalog_hysteresis' := '0.2'}
{attribute 'ac_datalog' := 'DatalogChannel'}
SP_MC_controller : REAL;
{attribute 'ac_datalog_hysteresis' := '2'}
{attribute 'ac_datalog' := 'DatalogChannel'}
Prerotary_output : REAL;
{attribute 'ac_datalog_hysteresis' := '2'}
{attribute 'ac_datalog' := 'DatalogChannel'}
VGD_output : REAL;
{attribute 'ac_datalog_hysteresis' := '2'}
{attribute 'ac_datalog' := 'DatalogChannel'}
SP_PID_compressor : REAL;
{attribute 'ac_datalog_hysteresis' := '2'}
{attribute 'ac_datalog' := 'DatalogChannel'}
Output_PID_suction : REAL;
{attribute 'ac_datalog_hysteresis' := '2'}
{attribute 'ac_datalog' := 'DatalogChannel'}
Output_PID_discharge : REAL;
{attribute 'ac_datalog_hysteresis' := '2'}
{attribute 'ac_datalog' := 'DatalogChannel'}
Output_PID_motor : REAL;
{attribute 'ac_datalog_hysteresis' := '2'}
{attribute 'ac_datalog' := 'DatalogChannel'}
Output_PID_superheat : REAL;
{attribute 'ac_datalog_hysteresis' := '2'}
{attribute 'ac_datalog' := 'DatalogChannel'}
SP_control : REAL;
{attribute 'ac_datalog_hysteresis' := '2'}
{attribute 'ac_datalog' := 'DatalogChannel'}
Unit_control_signal : REAL;
{attribute 'ac_datalog_hysteresis' := '2'}
{attribute 'ac_datalog' := 'DatalogChannel'}
Feedback_PRV : REAL;
{attribute 'ac_datalog_hysteresis' := '0.3'}
{attribute 'ac_datalog' := 'DatalogChannel'}
Theta_out : REAL;
{attribute 'ac_datalog_hysteresis' := '50'}
{attribute 'ac_datalog' := 'DatalogChannel'}
Alarm_limit_stall_count_unscaled : WORD;
{attribute 'ac_datalog_hysteresis' := '50'}
{attribute 'ac_datalog' := 'DatalogChannel'}
Alarm_limit_stall_count : REAL;
{attribute 'ac_datalog_hysteresis' := '2'}
{attribute 'ac_datalog' := 'DatalogChannel'}
Stall_ramp : REAL;
Min_allowed_PRVposition : REAL;
Number_of_starts : REAL;
SP_oil_pressure : REAL;
{attribute 'ac_datalog_hysteresis' := '2'}
{attribute 'ac_datalog' := 'DatalogChannel'}
Setpoint_conv_oil_pump : REAL;
Days_above_stall_limit : REAL;
Hrs_above_stall_limit : REAL;
Min_above_stall_limit : REAL;
Sec_above_stall_limit : REAL;
{attribute 'ac_datalog_hysteresis' := '2'}
{attribute 'ac_datalog' := 'DatalogChannel'}
SP_cond_press : REAL;
{attribute 'ac_datalog_hysteresis' := '2'}
{attribute 'ac_datalog' := 'DatalogChannel'}
SP_PID_Level : REAL;
{attribute 'ac_datalog_hysteresis' := '2'}
{attribute 'ac_datalog' := 'DatalogChannel'}
Control_signal_SW_valve : REAL;
{attribute 'ac_datalog_hysteresis' := '4'}
{attribute 'ac_datalog' := 'DatalogChannel'}
Liquid_valve_output : REAL;
{attribute 'ac_datalog_hysteresis' := '0.2'}
{attribute 'ac_datalog' := 'DatalogChannel'}
SP_PID_seawater : REAL;
{attribute 'ac_datalog_hysteresis' := '4'}
{attribute 'ac_datalog' := 'DatalogChannel'}
Chiller_capacity_t1 : REAL;
{attribute 'ac_datalog_hysteresis' := '2'}
{attribute 'ac_datalog' := 'DatalogChannel'}
SW_pump_speed_order : REAL;
{attribute 'ac_datalog_hysteresis' := '0.4'}
{attribute 'ac_datalog' := 'DatalogChannel'}
Press_chilled_medium_out : REAL;
{attribute 'ac_datalog_hysteresis' := '50'}
{attribute 'ac_datalog' := 'DatalogChannel'}
Running_hours_compressormotor : REAL;
{attribute 'ac_datalog_hysteresis' := '0.2'}
{attribute 'ac_datalog' := 'DatalogChannel'}
Press_water_cond_inlet : REAL;
{attribute 'ac_datalog_hysteresis' := '2'}
{attribute 'ac_datalog' := 'DatalogChannel'}
Speed_feedback_VFD : REAL;
{attribute 'ac_datalog_hysteresis' := '2'}
{attribute 'ac_datalog' := 'DatalogChannel'}
Order_VFD_perc : REAL;
{attribute 'ac_datalog_hysteresis' := '2'}
{attribute 'ac_datalog' := 'DatalogChannel'}
Order_VFD_Hz : REAL;
{attribute 'ac_datalog_hysteresis' := '2'}
{attribute 'ac_datalog' := 'DatalogChannel'}
Temp_trafo_wind_U : REAL;
{attribute 'ac_datalog_hysteresis' := '0.2'}
{attribute 'ac_datalog' := 'DatalogChannel'}
Temp_trafo_wind_V : REAL;
{attribute 'ac_datalog_hysteresis' := '0.2'}
{attribute 'ac_datalog' := 'DatalogChannel'}
Temp_trafo_wind_W : REAL;
{attribute 'ac_datalog_hysteresis' := '2'}
{attribute 'ac_datalog' := 'DatalogChannel'}
Opt_speed_VFD_perc : REAL;
{attribute 'ac_datalog_hysteresis' := '2'}
{attribute 'ac_datalog' := 'DatalogChannel'}
Opt_speed_VFD_Hz : REAL;
Surge_counter_VFD : REAL;
Spare_4 : REAL;
Spare_3 : REAL;
Spare_2 : REAL;
Spare_0 : REAL;
Vibration_compressor_DE: REAL;
Vibration_compressor_NDE: REAL;
Feedback_seawater_valve_overboard : REAL;
Feedback_seawater_valve_bypass : REAL;
CW_flow_m3: REAL;
SW_flow_m3: REAL;
Max_motor_wind_temp: REAL;
Order_SWW_overboard: REAL;
Order_SWW_bypass: REAL;
{attribute 'ac_datalog_hysteresis' := '0.4'}
{attribute 'ac_datalog' := 'DatalogChannel_4'}
COP_chiller_mech : REAL ;
{attribute 'ac_datalog_hysteresis' := '10'}
{attribute 'ac_datalog' := 'DatalogChannel_4'}
P2_mot_1_kW : REAL ;
{attribute 'ac_datalog_hysteresis' := '20'}
{attribute 'ac_datalog' := 'DatalogChannel_4'}
P1_motor_kW : REAL ;
{attribute 'ac_datalog_hysteresis' := '0.4'}
{attribute 'ac_datalog' := 'DatalogChannel_4'}
COP_chiller_ele : REAL ;
{attribute 'ac_datalog_hysteresis' := '0.2'}
{attribute 'ac_datalog' := 'DatalogChannel_4'}
PI_chiller : REAL ;
;{attribute 'ac_datalog_hysteresis' := '40'}
{attribute 'ac_datalog' := 'DatalogChannel_4'}
Wasted_energy_kW : REAL ;
{attribute 'ac_datalog_hysteresis' := '200'}
{attribute 'ac_datalog' := 'DatalogChannel'}
Chiller_capacity_kW : REAL;
Thrust_bearing_ref_min : REAL ;
Thrust_bearing_ref_max : REAL ;
Thrust_bearing_ref : REAL ;
Q2_chillerMWh : REAL ;
Chiller_P1_MWh : REAL ;
Cal_date_MMYY : REAL ;
Chiller_P2_MWh : REAL ;
Refrigerant_liquid_temp : REAL ;
VFD_motor_current : REAL ;
Feedback_liquid_valve_raw : REAL ;
Feedback_VGD_raw : REAL ;
Feedback_PRV_raw : REAL ;
Feedback_HGV_raw : REAL ;
Feedback_seawater_valve_overboard_raw : REAL ;
Feedback_seawater_valve_bypass_raw : REAL ;
SP_cond_press_limit : REAL ;
SP_evap_press_limit : REAL ;
SP_discharge_superheat_limit : REAL ;
VFD_min_allowed_frequence : REAL ;
VFD_min_allowed_speed : REAL ;

Trip_BITs_0_to_15 : WORD;
Trip_BITs_16_to_31: WORD;
Trip_BITs_32_to_47: WORD;
Trip_BITs_48_to_63: WORD;
Trip_BITs_64_to_79: WORD;
Trip_BITs_80_to_95: WORD;
Trip_BITs_96_to_121: WORD;
Trip_BITs_122_to_137: WORD;
Trip_BITs_138_to_153: WORD;
Trip_BITs_154_to_169: WORD;
Trip_BITs_170_to_185: WORD;
Trip_BITs_186_to_201: WORD;


Alarm_BITs_0_to_15: WORD;
Alarm_BITs_16_to_31: WORD;
Alarm_BITs_32_to_47: WORD;
Alarm_BITs_48_to_63: WORD;
Alarm_BITs_64_to_79: WORD;
Alarm_BITs_80_to_95: WORD;
Alarm_BITs_96_to_111: WORD;
Statusbits_0_to_15 : WORD;
Statusbits_16_to_31 : WORD;
Statusbits_32_to_47: WORD;
Statusbits_48_to_63: WORD;
Statusbits_64_to_79: WORD;
Statusbits_80_to_95: WORD;




DIStatusbits_0_to_15 : WORD;
DIStatusbits_16_to_31: WORD;

DOStatusbits_16_to_31: WORD;
DOStatusbits_32_to_47: WORD;

T_Overload_compressor_motor : BOOL;
T_Compressor_running_failure : BOOL;

T_Low_oil_flow : BOOL;
T_Overload_oil_pump_motor : BOOL;
T_Oil_pump_running_failure : BOOL;
T_Low_oil_flow_trip : BOOL;
T_High_temp_oil_receiver : BOOL;
T_Low_temp_oil_receiver : BOOL;
T_Low_suction_pressure : BOOL;
T_High_suction_pressure : BOOL;
T_High_discharge_pressure : BOOL;
T_Low_discharge_pressure : BOOL;
T_High_discharge_temp : BOOL;
T_Low_oil_diff_pressure : BOOL;
T_High_diff_oil_pressure : BOOL;
T_Starting_to_long : BOOL;
T_Surge_detection : BOOL;
T_Comp_thrust_bearing_position : BOOL;
Spare_trip_1 : BOOL;
T_Chilled_pump_run_failure : BOOL;
T_Sea_water_pump_run_failure : BOOL;
T_Low_chilled_medium_flow : BOOL;
T_High_chilled_medium_flow : BOOL;
T_Low_condenser_flow : BOOL;
T_High_condenser_flow : BOOL;
T_Emergency_stop : BOOL;
T_High_comp_mot_DE_bear_temp : BOOL;
T_High_comp_mot_NDE_bear_temp : BOOL;
T_High_motor_air_temp : BOOL;
T_Comp_motor_leak_detection : BOOL;
T_High_comp_mot_DE_bear_vib : BOOL;
T_High_comp_mot_NDE_bear_Vib : BOOL;
Spare_trip_2 : BOOL;
T_Rotating_stall_trip : BOOL;
T_Analog_inputs : BOOL;
T_Feedback_CW_valve : BOOL;
T_Low_oil_diff_press_prelub : BOOL;
T_Low_oil_diff_press_standstil : BOOL;

T_Spare_3 : BOOL;
T_Spare_4 : BOOL;
T_Spare_5 : BOOL;
T_Spare_6 : BOOL;
T_Spare_7 : BOOL;
T_Spare_8 : BOOL;
T_High_temp_oil_inlet_comp : BOOL;
T_Comp_motor_power_loss : BOOL;
Spare_trip_3 : BOOL;
T_Cathodic_protect_sys_alarm : BOOL;
T_High_oil_filter_diff_press : BOOL;
T_Flow_switch_FT01 : BOOL;
T_Starter_failure_trip : BOOL;
T_Incorrect_feedback_starter_trip : BOOL;


A_High_condenser_flow : BOOL;
A_Rotating_stall : BOOL;
A_High_temp_oil_inlet_comp : BOOL;
SpareAlarm_1 : BOOL;
A_High_motor_air_temp : BOOL;
A_High_control_panel_temp : BOOL;
A_Low_oil_diff_pressure : BOOL;
Spare_alarm_2 : BOOL;
A_High_comp_motor_winding_temp : BOOL;
A_High_comp_mo_DE_bear_temp : BOOL;
A_High_comp_mo_NDE_bear_temp : BOOL;
A_High_comp_mo_DE_bear_vib : BOOL;
A_High_comp_mo_NDE_bear_vib : BOOL;
A_Low_chilled_medium_flow : BOOL;
A_High_chilled_medium_flow : BOOL;
A_Low_sea_water_flow : BOOL;
A_Seawater_pump_not_running : BOOL;
A_Spare : BOOL;
A_Spare_1 : BOOL;
A_Spare_2 : BOOL;
A_Spare_3 : BOOL;
A_Spare_4 : BOOL;
A_Spare_5 : BOOL;
A_Spare_6 : BOOL;
A_Spare_7 : BOOL;
A_Spare_8 : BOOL;
A_Spare_9 : BOOL;
A_Spare_10 : BOOL;
A_Spare_11 : BOOL;
A_High_oil_filter_diff_press : BOOL;
A_Spare_12 : BOOL;
A_Spare_13 : BOOL;
A_Spare_14 : BOOL;
A_Spare_15 : BOOL;
A_Spare_16 : BOOL;
A_Spare_17 : BOOL;
Anti_recycle_status : BOOL;
Low_oil_temperature : BOOL;
Low_oil_temp_auto : BOOL;
Oil_heater : BOOL;
Sea_water_pump : BOOL;
Comp_oil_pump : BOOL;
Bearing_oil_pump : BOOL;
Solenoid_oil_return : BOOL;
Unit_running : BOOL;
Unit_remote : BOOL;
Unit_auto : BOOL;
Unit_manual : BOOL;
Unit_trip : BOOL;
Unit_alarm : BOOL;
Unit_start_switch : BOOL;
Unit_avabiable : BOOL;
S_Spare_1 : BOOL;
S_Spare_2 : BOOL;
S_Spare_3 : BOOL;
S_Spare_4 : BOOL;
S_Spare_5 : BOOL;
S_Spare_6 : BOOL;
S_Spare_7 : BOOL;
S_Spare_8 : BOOL;
Solenoid_liquid_inj: BOOL;
CW_Flow_ind : BOOL;
Open_chilled_water_valve : BOOL;
Feedback_chilled_water_valve : BOOL;
Open_order_swv_overboard : BOOL;
Close_order_swv_overboard : BOOL;
Open_order_swv_bypass : BOOL;
Close_order_swv_bypass : BOOL;
VFD_man_auto : BOOL ;
VFD_freq_jump_on : BOOL ;
VFD_ramp_100_perc : BOOL ;
VFD_locked_100_perc : BOOL;
VFD_ramp_d_PRVcontrol : BOOL;
PRV_control : BOOL;
VFD_control : BOOL;
Spare_151: BOOL;
T_Transformer_winding_temp : BOOL;
A_Transformer_winding_temp : BOOL;
T_trafo_opening_main_breaker : BOOL;
T_VFD : BOOL;
VFD_ready : BOOL;
T_VFD_emergency_stop : BOOL;
T_Low_5VDC_supply : BOOL;
T_High_5VDC_supply : BOOL;
T_Spare_9 : BOOL;
T_Spare_10 : BOOL;
T_Spare_11 : BOOL;
T_Spare_12 : BOOL;
T_Spare_13 : BOOL;
T_Low_liquid_level : BOOL;
T_SW_pump_off_to_long : BOOL;
T_Softstarter_failure : BOOL;
T_Motorstarter_failure : BOOL ;
T_CW_valveopen_failure : BOOL ;
T_SW_valveopen_failure : BOOL ;
T_High_disch_superheat :BOOL ;
T_Low_disch_superheat :BOOL ;
T_High_CW_outlet_temp : BOOL;
T_Low_CW_outlet_temp : BOOL;
T_Low_CW_inlet_temp : BOOL;
T_High_CW_inlet_temp : BOOL;
T_High_SW_outlet_temp : BOOL;
T_Low_SW_outlet_temp : BOOL;
T_Low_SW_inlet_temp : BOOL;
T_High_SW_inlet_temp : BOOL;
T_High_motor_wind_temp_R : BOOL;
T_High_motor_wind_temp_S : BOOL;
T_High_motor_wind_temp_T : BOOL;
T_High_motor_wind_temp : BOOL;
T_High_press_ratio : BOOL;
T_Low_press_ratio : BOOL;
T_Low_CW_dP : BOOL;
T_High_CW_dP : BOOL;
T_Low_SW_dP : BOOL;
T_High_SW_dP : BOOL;
T_Long_time_PRV : BOOL;
T_Comp_thrust_neg_move : BOOL;
T_Comp_thrust_pos_move : BOOL;
T_VGD_fault : BOOL;
T_Low_oilpress_prelube : BOOL;
T_Low_temp_oil_inlet_comp : BOOL;
T_Low_oilpress_standby : BOOL;


T_Sensor_high_signal_AI_64 : BOOL;
T_Sensor_low_signal_AI_64 : BOOL ;
T_Sensor_high_signal_AI_66 : BOOL;
T_Sensor_low_signal_AI_66 : BOOL ;
T_Sensor_high_signal_AI_128 : BOOL;
T_Sensor_low_signal_AI_128 : BOOL ;
T_Sensor_high_signal_AI_130 : BOOL;
T_Sensor_low_signal_AI_130 : BOOL ;
T_Sensor_high_signal_AI_132 : BOOL;
T_Sensor_low_signal_AI_132 : BOOL ;
T_Sensor_high_signal_AI_134 : BOOL;
T_Sensor_low_signal_AI_134 : BOOL ;
T_Sensor_high_signal_AI_136 : BOOL;
T_Sensor_low_signal_AI_136 : BOOL ;
T_Sensor_high_signal_AI_138 : BOOL;
T_Sensor_low_signal_AI_138 : BOOL ;
T_Sensor_high_signal_AI_140 : BOOL;
T_Sensor_low_signal_AI_140 : BOOL ;
T_Sensor_high_signal_AI_142 : BOOL;
T_Sensor_low_signal_AI_142 : BOOL ;
T_Sensor_high_signal_AI_144 : BOOL;
T_Sensor_low_signal_AI_144 : BOOL ;
T_Sensor_high_signal_AI_146 : BOOL;
T_Sensor_low_signal_AI_146 : BOOL ;
T_Sensor_high_signal_AI_148 : BOOL;
T_Sensor_low_signal_AI_148 : BOOL ;
T_Sensor_high_signal_AI_150 : BOOL;
T_Sensor_low_signal_AI_150 : BOOL ;
T_Sensor_high_signal_AI_152 : BOOL;
T_Sensor_low_signal_AI_152 : BOOL ;
T_Sensor_high_signal_AI_154 : BOOL;
T_Sensor_low_signal_AI_154 : BOOL ;
T_Sensor_high_signal_AI_156 : BOOL;
T_Sensor_low_signal_AI_156 : BOOL ;
T_Sensor_high_signal_AI_158 : BOOL;
T_Sensor_low_signal_AI_158 : BOOL ;
T_Sensor_high_signal_AI_160 : BOOL;
T_Sensor_low_signal_AI_160 : BOOL ;
T_Sensor_high_signal_AI_162 : BOOL;
T_Sensor_low_signal_AI_162 : BOOL ;
T_Sensor_high_signal_AI_164 : BOOL;
T_Sensor_low_signal_AI_164 : BOOL ;
T_Sensor_high_signal_AI_166 : BOOL;
T_Sensor_low_signal_AI_166 : BOOL ;
T_Sensor_high_signal_AI_168 : BOOL;
T_Sensor_low_signal_AI_168 : BOOL ;
T_Sensor_high_signal_AI_170 : BOOL;
T_Sensor_low_signal_AI_170 : BOOL ;
T_Sensor_high_signal_AI_172 : BOOL;
T_Sensor_low_signal_AI_172 : BOOL ;
T_Sensor_high_signal_AI_174 : BOOL;
T_Sensor_low_signal_AI_174 : BOOL ;
T_Sensor_high_signal_AI_176 : BOOL;
T_Sensor_low_signal_AI_176 : BOOL ;
T_Sensor_low_signal_AI_178 : BOOL ;
T_Sensor_high_signal_AI_178 : BOOL;
T_Sensor_low_signal_AI_180 : BOOL ;
T_Sensor_high_signal_AI_180 : BOOL;
T_Sensor_low_signal_AI_182 : BOOL ;
T_Sensor_high_signal_AI_182 : BOOL;
T_Sensor_low_signal_AI_184 : BOOL ;
T_Sensor_high_signal_AI_184 : BOOL;
T_Sensor_low_signal_AI_186 : BOOL ;
T_Sensor_high_signal_AI_186 : BOOL;
T_Sensor_low_signal_AI_188 : BOOL ;
T_Sensor_high_signal_AI_188 : BOOL;
T_Sensor_low_signal_AI_190 : BOOL ;
T_Sensor_high_signal_AI_190 : BOOL;
T_Sensor_low_signal_AI_192 : BOOL ;
T_Sensor_high_signal_AI_192 : BOOL;
T_Sensor_low_signal_AI_194 : BOOL ;
T_Sensor_high_signal_AI_194 : BOOL;
T_Sensor_low_signal_AI_196 : BOOL ;
T_Sensor_high_signal_AI_196 : BOOL;
T_Sensor_low_signal_AI_198 : BOOL ;
T_Sensor_high_signal_AI_198 : BOOL;
T_Sensor_high_signal_AI_200 : BOOL;
T_Sensor_low_signal_AI_200 : BOOL ;
T_Sensor_low_signal_AI_202 : BOOL ;
T_Sensor_high_signal_AI_202 : BOOL;
T_Sensor_low_signal_AI_204 : BOOL ;
T_Sensor_high_signal_AI_204 : BOOL;
T_Sensor_low_signal_AI_206 : BOOL ;
T_Sensor_high_signal_AI_206 : BOOL ;
T_Sensor_signal_5VDC_supply  : BOOL ;
T_Sensor_signal_Motor_current  : BOOL ;
T_Sensor_signal_PRV_position  : BOOL ;
T_Sensor_signal_CW_inlet_temp  : BOOL ;
T_Sensor_signal_HGV_position  : BOOL ;
T_Sensor_signal_suction_press  : BOOL ;
T_Sensor_signal_discharge_press  : BOOL ;
T_Sensor_signal_oil_press_receiver  : BOOL ;
T_Sensor_signal_oil_compr  : BOOL ;
T_Sensor_signal_discharge_temp  : BOOL ;
T_Sensor_signal_oil_receiver_temp  : BOOL ;
T_Sensor_signal_CW_outlet_temp  : BOOL ;
T_Sensor_signal_thrust_bearing_pos  : BOOL ;

T_Sensor_signal_SW_press_inlet  : BOOL ;
T_Sensor_signal_SW_press_outlet  : BOOL ;
T_Sensor_signal_SW_temp_inlet  : BOOL ;
T_Sensor_signal_SW_temp_outlet  : BOOL ;
T_Sensor_signal_motor_air_temp  : BOOL ;
T_Sensor_signal_temp_motor_wind_R  : BOOL ;
T_Sensor_signal_temp_motor_wind_S  : BOOL ;
T_Sensor_signal_temp_motor_wind_T  : BOOL ;
T_Sensor_signal_comp_mot_DE_bear_temp  : BOOL ;
T_Sensor_signal_comp_mot_NDE_bear_temp : BOOL ;



A_high_disch_press : BOOL ;
A_low_disch_press : BOOL ;
A_Low_suction_pressure : BOOL;
A_High_suction_pressure : BOOL;
A_High_discharge_temp : BOOL;
A_High_oil_temp_receiver : BOOL;
A_Low_oil_temp_receiver : BOOL;
A_Low_temp_oil_inlet_comp : BOOL;
A_High_oil_diff_pressure : BOOL;
A_Low_discharge_superheat : BOOL;
A_High_discharge_superheat : BOOL;
A_Low_CW_outlet_temp : BOOL;
A_High_CW_outlet_temp : BOOL;
A_Low_CW_inlet_temp : BOOL;
A_High_CW_inlet_temp : BOOL;
A_High_SW_outlet_temp : BOOL;
A_Low_condenser_flow : BOOL;
A_High_press_ratio : BOOL;
A_Low_press_ratio : BOOL;
A_Motor_speed_low : BOOL;
A_Low_SW_outlet_temp : BOOL;
A_Low_SW_inlet_temp : BOOL;
A_High_SW_inlet_temp : BOOL;
A_High_suction_superheat : BOOL;
A_Low_suction_superheat : BOOL;
A_High_temp_oil_separator : BOOL;
A_Low_temp_oil_separator : BOOL;
A_High_motor_wind_temp_R : BOOL;
A_High_motor_wind_temp_S : BOOL;
A_High_motor_wind_temp_T : BOOL;
A_High_motor_wind_temp : BOOL;
A_High_CW_dP : BOOL;
A_Low_CW_dP : BOOL;
A_High_SW_dP : BOOL;
A_Low_SW_dP : BOOL;
A_VGD_Fault : BOOL;
Start_inhib_time_between_Start : BOOL;
Start_inhib_time_beetween_Stop : BOOL;
Start_inhib_PRV_not_min : BOOL;
Start_inhib_Motor_overload : BOOL;
Remote_bilge_pump_control : BOOL;
CW_pump_running : BOOL;
A_Low_liquid_level : BOOL;
A_Suction_press_limit : BOOL;
A_Discharge_press_limit : BOOL;
A_Discharge_superheat_limit : BOOL;
A_Motor_current_limit : BOOL;
A_Backup_battery : BOOL; 
A_Temp_motor_bearing_NDE : BOOL;
A_Temp_motor_bearing_DE : BOOL;

DI_0_0_Emergency_stop : BOOL;
DI_0_1 : BOOL;
DI_0_2_Fault_reset : BOOL;
DI_0_3 : BOOL;
DI_0_4 : BOOL;
DI_0_5 : BOOL;
DI_0_6_Overload_protection : BOOL;
DI_0_7 : BOOL;
DI_1_0_Overload_oilpump : BOOL;
DI_1_1 : BOOL;
DI_1_2 : BOOL;
DI_1_3 : BOOL;
DI_1_4_Power_availible : BOOL;
DI_1_5_Starter_failure : BOOL;
DI_8_0_Controlpanel_temp : BOOL;
DI_8_1 : BOOL;
DI_8_2_VGD_limit_switch : BOOL;
DI_8_3_water_leak_motor  : BOOL;
DI_8_4_Catodic_protection : BOOL;
DI_8_5_Trust_bearing_probe : BOOL;
DI_8_6_ESD_operation : BOOL;
DI_8_7 : BOOL;
DI_9_0_MV_breaker_availible : BOOL;
DI_9_1 : BOOL;
DI_9_2_Safe_return_to_port : BOOL;
DI_9_3 : BOOL;
DI_9_4_VFD_emergency_stop : BOOL;
DI_9_5 : BOOL;
DI_9_6 : BOOL;
DI_9_7 : BOOL;
DO_0_0 : BOOL;
DO_0_1 : BOOL;
DO_0_2 : BOOL;
DO_0_3 : BOOL;
DO_0_4 : BOOL;
DO_0_5 : BOOL;
DO_0_6 : BOOL;
DO_0_7 : BOOL;
DO_1_0 : BOOL;
DO_1_1 : BOOL;
DO_8_0 : BOOL;
DO_8_1 : BOOL;
DO_8_2 : BOOL;
DO_8_3 : BOOL;
DO_8_4 : BOOL;
DO_8_5 : BOOL;
DO_8_6 : BOOL;
DO_8_7 : BOOL;
DO_9_0 : BOOL;
DO_9_1 : BOOL;
DO_9_2 : BOOL;
DO_9_3 : BOOL;
DO_9_4 : BOOL;
DO_9_5 : BOOL;
DO_9_6 : BOOL;
DO_9_7 : BOOL;
DO_12_0 : BOOL;
DO_12_1 : BOOL;
DO_12_2 : BOOL;
DO_12_3 : BOOL;
DO_12_4 : BOOL;
DO_12_5 : BOOL;
DO_12_6 : BOOL;
DO_12_7 : BOOL;



//Graphic variables
Unit_switch_status : INT;
i : INT;
show_trendvalue : ARRAY[0..50] OF BOOL;
select_trendvalue : INT :=0 ;

END_VAR


modbus_var[0] :=%IW0;
Temp_chilled_medium_out:=scaleFunction(modbus_var_1000[21],0.1, 0);
Temp_chilled_medium_in:=scaleFunction(modbus_var_1000[22],0.1, 0);
Temp_water_inlet_cond:=scaleFunction(modbus_var_1000[23],0.1, 0);
Press_suction_compr:=scaleFunction(modbus_var_1000[24],0.01, 0);
Press_discharge_compr:=scaleFunction(modbus_var_1000[25],0.01, 0);
Oil_diff_pressure:=scaleFunction(modbus_var_1000[26],0.01, 0);
Suction_saturated_temp:=scaleFunction(modbus_var_1000[27],0.01, 0);
Temp_discharge:=scaleFunction(modbus_var_1000[28],0.1, 0);
Oil_temp_receiver:=scaleFunction(modbus_var_1000[29],0.1, 0);
Press_oil_receiver:=scaleFunction(modbus_var_1000[30],1.0, 0);
Press_oil_compr:=scaleFunction(modbus_var_1000[31],0.1, 0);
SP_CW_controller:=scaleFunction(modbus_var_1000[32],0.1, 0);
Motor_current:=scaleFunction(modbus_var_1000[33],0.1, 0);

// convert running hours compressor
Running_hours_comp_unscaled:=modbus_var_1000[34];
Running_hours_compressormotor:=Running_hours_comp_unscaled*1.0;

Anti_recycle_time:=scaleFunction(modbus_var_1000[35],1.0, 0);
Feedback_PRV:=scaleFunction(modbus_var_1000[36],0.1, 0);
spare:=scaleFunction(modbus_var_1000[37],0.01, 0);
dP_SW:=scaleFunction(modbus_var_1000[38],0.1, 0);
Temp_motor_bearing_DE:=scaleFunction(modbus_var_1000[39],0.1, 0);
Temp_motor_bearing_NDE:=scaleFunction(modbus_var_1000[40],0.1, 0);
Temp_motor_wind_R:=scaleFunction(modbus_var_1000[41],0.1, 0);
Temp_motor_wind_S:=scaleFunction(modbus_var_1000[42],0.1, 0);
Temp_motor_wind_T:=scaleFunction(modbus_var_1000[43],0.1, 0);
Max_motor_temp:=scaleFunction(modbus_var_1000[44],0.1, 0);
Temp_motor_air:=scaleFunction(modbus_var_1000[45],0.01, 0);
spare:=scaleFunction(modbus_var_1000[46],0.01, 0);
spare:=scaleFunction(modbus_var_1000[47],0.1, 0);
Chiller_capacity:=scaleFunction(modbus_var_1000[48],0.1, 0);
Temp_water_outlet_cond:=scaleFunction(modbus_var_1000[49],1.0, 0);
Feedback_liquid_valve:=scaleFunction(modbus_var_1000[50],0.1, 0);
Feedback_HGV:=scaleFunction(modbus_var_1000[51],0.01, 0);
Press_water_cond_out:=scaleFunction(modbus_var_1000[52],0.1, 0);
Press_water_cond_inlet:=scaleFunction(modbus_var_1000[53],0.1, 0);
Liquid_level_condenser:=scaleFunction(modbus_var_1000[54],0.1, 0);
SP_PID_seawater:=scaleFunction(modbus_var_1000[55],0.1, 0);
Discharge_superheat:=scaleFunction(modbus_var_1000[56],0.1, 0);
spare:=scaleFunction(modbus_var_1000[57],0.01, 0);
Discharge_saturated_temp:=scaleFunction(modbus_var_1000[58],0.1, 0);

// Calculation theta out
Theta_out:=Temp_chilled_medium_out-Suction_saturated_temp;



Trip_BITs_0_to_15:=modbus_var_1000[0];
Trip_BITs_16_to_31:=modbus_var_1000[1];
Trip_BITs_32_to_47:=modbus_var_1000[2];
Trip_BITs_48_to_63:=modbus_var_1000[3];
Trip_BITs_64_to_79:=modbus_var_1000[4];
Alarm_BITs_0_to_15:=modbus_var_1000[5];
Statusbits_0_to_15:=modbus_var_1000[6];
Statusbits_16_to_31:=modbus_var_1000[7];


// Trip bits
T_Overload_compressor_motor:=maskbitFunction(Trip_BITs_0_to_15,0);
T_Compressor_running_failure:=maskbitFunction(Trip_BITs_0_to_15,1);
T_Low_CW_outlet_temp:=maskbitFunction(Trip_BITs_0_to_15,2);
T_Low_oil_flow:=maskbitFunction(Trip_BITs_0_to_15,3);
T_Overload_oil_pump_motor:=maskbitFunction(Trip_BITs_0_to_15,4);
T_Oil_pump_running_failure:=maskbitFunction(Trip_BITs_0_to_15,5);
T_Low_oil_flow_trip:=maskbitFunction(Trip_BITs_0_to_15,6);
T_High_temp_oil_receiver:=maskbitFunction(Trip_BITs_0_to_15,7);
T_Low_suction_pressure:=maskbitFunction(Trip_BITs_0_to_15,8);
T_High_discharge_pressure:=maskbitFunction(Trip_BITs_0_to_15,9);
T_High_discharge_temp:=maskbitFunction(Trip_BITs_0_to_15,10);
T_Low_oil_diff_pressure:=maskbitFunction(Trip_BITs_0_to_15,11);
T_High_diff_oil_pressure:=maskbitFunction(Trip_BITs_0_to_15,12);
T_Starting_to_long:=maskbitFunction(Trip_BITs_0_to_15,13);
T_Surge_detection:=maskbitFunction(Trip_BITs_0_to_15,14);
T_Comp_thrust_bearing_position:=maskbitFunction(Trip_BITs_0_to_15,15);
T_High_5VDC_supply:=maskbitFunction(Trip_BITs_16_to_31,0);
T_Chilled_pump_run_failure:=maskbitFunction(Trip_BITs_16_to_31,1);
T_Sea_water_pump_run_failure:=maskbitFunction(Trip_BITs_16_to_31,2);
S_Spare_1:=maskbitFunction(Trip_BITs_16_to_31,3);
S_Spare_1:=maskbitFunction(Trip_BITs_16_to_31,4);
T_Low_SW_dP:=maskbitFunction(Trip_BITs_16_to_31,5);
T_High_SW_dP:=maskbitFunction(Trip_BITs_16_to_31,6);
T_Emergency_stop:=maskbitFunction(Trip_BITs_16_to_31,7);
T_High_motor_wind_temp:=maskbitFunction(Trip_BITs_16_to_31,8);
T_High_comp_mot_DE_bear_temp:=maskbitFunction(Trip_BITs_16_to_31,9);
T_High_comp_mot_NDE_bear_temp:=maskbitFunction(Trip_BITs_16_to_31,10);
T_High_motor_air_temp:=maskbitFunction(Trip_BITs_16_to_31,11);
T_Comp_motor_leak_detection:=maskbitFunction(Trip_BITs_16_to_31,12);
S_Spare_1:=maskbitFunction(Trip_BITs_16_to_31,13);
S_Spare_1:=maskbitFunction(Trip_BITs_16_to_31,14);
T_Low_5VDC_supply:=maskbitFunction(Trip_BITs_16_to_31,15);
T_Sensor_signal_5VDC_supply:=maskbitFunction(Trip_BITs_32_to_47,0);
T_Sensor_signal_Motor_current:=maskbitFunction(Trip_BITs_32_to_47,1);
T_Sensor_signal_PRV_position:=maskbitFunction(Trip_BITs_32_to_47,2);
T_Sensor_signal_CW_inlet_temp:=maskbitFunction(Trip_BITs_32_to_47,3);
T_Sensor_signal_HGV_position:=maskbitFunction(Trip_BITs_32_to_47,4);
T_Spare_6:=maskbitFunction(Trip_BITs_32_to_47,5);
T_Spare_7:=maskbitFunction(Trip_BITs_32_to_47,6);
T_Spare_8:=maskbitFunction(Trip_BITs_32_to_47,7);
T_Sensor_signal_suction_press:=maskbitFunction(Trip_BITs_32_to_47,8);
T_Sensor_signal_discharge_press:=maskbitFunction(Trip_BITs_32_to_47,9);
T_Sensor_signal_oil_press_receiver:=maskbitFunction(Trip_BITs_32_to_47,10);
T_Sensor_signal_oil_compr:=maskbitFunction(Trip_BITs_32_to_47,11);
T_Sensor_signal_discharge_temp:=maskbitFunction(Trip_BITs_32_to_47,12);
T_Sensor_signal_oil_receiver_temp:=maskbitFunction(Trip_BITs_32_to_47,13);
T_Sensor_signal_CW_outlet_temp:=maskbitFunction(Trip_BITs_32_to_47,14);
T_Sensor_signal_thrust_bearing_pos:=maskbitFunction(Trip_BITs_32_to_47,15);
S_Spare_1:=maskbitFunction(Trip_BITs_48_to_63,0);
S_Spare_1:=maskbitFunction(Trip_BITs_48_to_63,1);
T_Sensor_signal_SW_press_inlet:=maskbitFunction(Trip_BITs_48_to_63,2);
T_Sensor_signal_SW_press_outlet:=maskbitFunction(Trip_BITs_48_to_63,3);
T_Sensor_signal_SW_temp_inlet:=maskbitFunction(Trip_BITs_48_to_63,4);
T_Sensor_signal_SW_temp_outlet:=maskbitFunction(Trip_BITs_48_to_63,5);
S_Spare_1:=maskbitFunction(Trip_BITs_48_to_63,6);
S_Spare_1:=maskbitFunction(Trip_BITs_48_to_63,7);
T_Sensor_signal_motor_air_temp:=maskbitFunction(Trip_BITs_48_to_63,8);
T_Sensor_signal_temp_motor_wind_R:=maskbitFunction(Trip_BITs_48_to_63,9);
T_Sensor_signal_temp_motor_wind_S:=maskbitFunction(Trip_BITs_48_to_63,10);
T_Sensor_signal_temp_motor_wind_T:=maskbitFunction(Trip_BITs_48_to_63,11);
T_Sensor_signal_comp_mot_DE_bear_temp:=maskbitFunction(Trip_BITs_48_to_63,12);
T_Sensor_signal_comp_mot_NDE_bear_temp:=maskbitFunction(Trip_BITs_48_to_63,13);
S_Spare_1:=maskbitFunction(Trip_BITs_48_to_63,14);
S_Spare_1:=maskbitFunction(Trip_BITs_48_to_63,15);


//Alarm bits
A_High_condenser_flow:=maskbitFunction(Alarm_BITs_0_to_15,0);
SpareAlarm_1:=maskbitFunction(Alarm_BITs_0_to_15,1);
A_Low_liquid_level:=maskbitFunction(Alarm_BITs_0_to_15,2);
SpareAlarm_1:=maskbitFunction(Alarm_BITs_0_to_15,3);
SpareAlarm_1:=maskbitFunction(Alarm_BITs_0_to_15,4);
A_High_control_panel_temp:=maskbitFunction(Alarm_BITs_0_to_15,5);
SpareAlarm_1:=maskbitFunction(Alarm_BITs_0_to_15,6);
A_Backup_battery:=maskbitFunction(Alarm_BITs_0_to_15,7);
A_High_motor_wind_temp:=maskbitFunction(Alarm_BITs_0_to_15,8);
A_Temp_motor_bearing_DE:=maskbitFunction(Alarm_BITs_0_to_15,9);
A_Temp_motor_bearing_NDE:=maskbitFunction(Alarm_BITs_0_to_15,10);
SpareAlarm_1:=maskbitFunction(Alarm_BITs_0_to_15,11);
SpareAlarm_1:=maskbitFunction(Alarm_BITs_0_to_15,12);
SpareAlarm_1:=maskbitFunction(Alarm_BITs_0_to_15,13);
SpareAlarm_1:=maskbitFunction(Alarm_BITs_0_to_15,14);
A_Low_sea_water_flow:=maskbitFunction(Alarm_BITs_0_to_15,15);



// Status Bits
S_Spare_1:=maskbitFunction(Statusbits_0_to_15,0);
S_Spare_1:=maskbitFunction(Statusbits_0_to_15,1);
Start_inhib_PRV_not_min:=maskbitFunction(Statusbits_0_to_15,2);
Unit_trip:=maskbitFunction(Statusbits_0_to_15,3);
Unit_alarm:=maskbitFunction(Statusbits_0_to_15,4);
Unit_start_switch:=maskbitFunction(Statusbits_0_to_15,5);
CW_pump_running:=maskbitFunction(Statusbits_0_to_15,6);
Sea_water_pump:=maskbitFunction(Statusbits_0_to_15,7);
Unit_running:=maskbitFunction(Statusbits_0_to_15,8);
Unit_avabiable:=maskbitFunction(Statusbits_0_to_15,9);
Unit_remote:=maskbitFunction(Statusbits_0_to_15,10);
Unit_auto:=maskbitFunction(Statusbits_0_to_15,11);
Anti_recycle_status:=maskbitFunction(Statusbits_0_to_15,12);
S_Spare_1:=maskbitFunction(Statusbits_0_to_15,13);
S_Spare_1:=maskbitFunction(Statusbits_0_to_15,14);
S_Spare_1:=maskbitFunction(Statusbits_0_to_15,15);



// Graphic controls
IF Unit_remote THEN
	Unit_switch_status:=2;
ELSIF Unit_auto THEN 
	Unit_switch_status:=3;
ELSIF Unit_manual THEN 
	Unit_switch_status:=4;

END_IF ;	

IF select_trendvalue > 0 THEN
	show_trendvalue[select_trendvalue]:= TRUE;
ELSIF select_trendvalue = 0 THEN
	FOR i := 0 TO 50 DO
      show_trendvalue[i] := FALSE;
   	END_FOR
END_IF ;	
	
// timer2 (IN:= TRUE, PT:=T#5S);;
//	IF timer2_Q THEN
//		Temp_motor_bearing_DE := Temp_motor_bearing_DE +1;
//		Motor_current := Motor_current + 1 ;
//		Timer2(IN:= FALSE);
//	END_IF

END_PROGRAM

// Device/Application/Calculus
PROGRAM Calculus
VAR


// MWCC

NakW_chiller_3 : REAL ;
NakW_chiller_4 : REAL ;

COP_chiller_3 : REAL ;
COP_chiller_4 : REAL ;
NakW_chiller_5 : REAL ;
NakW_chiller_6 : REAL ;

COP_chiller_5 : REAL ;
COP_chiller_6 : REAL ;
{attribute 'ac_datalog_hysteresis' := '100'}
{attribute 'ac_datalog' := 'DatalogChannel_4'}
Tot_Power_motor : REAL ;
{attribute 'ac_datalog_hysteresis' := '300'}
{attribute 'ac_datalog' := 'DatalogChannel_4'}
Tot_Q2 : REAL ;
{attribute 'ac_datalog_hysteresis' := '100'}
{attribute 'ac_datalog' := 'DatalogChannel_4'}
Tot_Q2_MWh : REAL ;
{attribute 'ac_datalog_hysteresis' := '100'}
{attribute 'ac_datalog' := 'DatalogChannel_4'}
Tot_P1_MWh : REAL ;
Power_motor_3_kW : REAL ;
Power_motor_4_kW : REAL ;
Power_motor_5_kW : REAL ;
Power_motor_6_kW : REAL ;
Power_3_not_zero : REAL ;
Power_4_not_zero : REAL ;
Power_5_not_zero : REAL ;
Power_6_not_zero : REAL ;

// SE700
Q2kW_chiller_1 : REAL ;
Q2kW_chiller_2 : REAL ;
Chiller_1_dpCW_bar : REAL ;
Chiller_2_dpCW_bar : REAL ;
Chiller_1_SR_dpCW_bar : REAL ;
Chiller_2_SR_dpCW_bar : REAL ;
Power_motor_1_kW : REAL ;
Power_motor_2_kW : REAL ;
Power_1_not_zero : REAL ;
Power_2_not_zero : REAL ;
NakW_chiller_1 : REAL ;
NakW_chiller_2 : REAL ;
COP_chiller_1 : REAL ;
COP_chiller_2 : REAL ;



Power_3_not_zero_func: WORD := 100;
Power_4_not_zero_func :  WORD := 100;
COP_chiller_3_func :  WORD := 100;
COP_chiller_4_func :  WORD := 100;
Power_5_not_zero_func: WORD := 100;
Power_6_not_zero_func :  WORD := 100;
COP_chiller_5_func :  WORD := 100;
COP_chiller_6_func :  WORD := 100;
Tot_Power_motor_func :  WORD := 100;
Tot_Q2_func :  WORD := 100;
Tot_Q2_MWh_func :  WORD := 100;
Tot_Na_MWh_func :  WORD := 100;
Power_motor_3_kW_func :  WORD := 100;
Power_motor_4_kW_func :  WORD := 100;

// SE700

Man_Auto_Chiller_1_func :  WORD := 100;
Man_Auto_Chiller_2_func :  WORD := 100;
//SE700_Chiller_1_Modb|||VALISERR(LOCAL.MODBUS2.Chiller_2.Program_number);//
//SE700_Chiller_2_Modb|||VALISERR(LOCAL.MODBUS2.Chiller_2.Program_number);
Flow_factor_chiller1_func :  WORD := 100;
Flow_factor_chiller2_func :  WORD := 100;


SR_Nom_dP_bar_func :  WORD := 100;


Chiller_1_dT_func :  WORD := 100;
Chiller_2_dT_func :  WORD := 100;
Chiller_1_max_dT_func :  WORD := 100;
Chiller_2_max_dT_func :  WORD := 100;
Chiller_1_Capacity_func :  WORD := 100;
Chiller_2_Capacity_func :  WORD := 100;
Chiller_1_CapacitykW_func :  WORD := 100;
Chiller_2_CapacitykW_func :  WORD := 100;
Chiller_1_dpCW_bar_func :  WORD := 100;
Chiller_2_dpCW_bar_func :  WORD := 100;
Chiller_1_SR_dpCW_bar_func :  WORD := 100;
Chiller_2_SR_dpCW_bar_func :  WORD := 100;
Power_motor_1_kW_func :  WORD := 100;
Power_motor_2_kW_func :  WORD := 100;
Power_1_not_zero_func :  WORD := 100;
Power_2_not_zero_func :  WORD := 100;
COP_chiller_1_func :  WORD := 100;
COP_chiller_2_func :  WORD := 100;
Chiller_1_Capacity_corr_flow_factor_func :  WORD := 100;
Chiller_2_Capacity_corr_flow_factor_func :  WORD := 100;
// New Variables
PI_chiller_1  : REAL ;
PI_chiller_1_word : WORD ;
PI_Calc_Error_AC1 : BOOL ;
PI_chiller_2  : REAL ;
PI_chiller_2_word : WORD ;
PI_Calc_Error_AC2 : BOOL ;
PI_chiller_3  : REAL ;
PI_chiller_3_word : WORD ;
PI_Calc_Error_AC3 : BOOL ;
PI_chiller_4  : REAL ;
PI_chiller_4_word : WORD ;
PI_Calc_Error_AC4 : BOOL ;
PI_chiller_5  : REAL ;
PI_chiller_5_word : WORD ;
PI_Calc_Error_AC5 : BOOL ;
PI_chiller_6  : REAL ;
PI_chiller_6_word : WORD ;
PI_Calc_Error_AC6 : BOOL ;
delaytimer2 : TON ;	
resetbuttons : BOOL := FALSE  ;
COP_theo_AC1 :REAL ;	
COP_theo_AC2 :REAL ;
COP_theo_AC3 :REAL ;
COP_theo_AC4 :REAL ;
COP_theo_AC5 :REAL ;
COP_theo_AC6 :REAL ;
totRunningChillers : INT;
WastedEnergy_AC1 :REAL ;
WastedEnergy_AC1_word :WORD ;
WastedEnergy_AC2 :REAL ;
WastedEnergy_AC2_word :WORD ;
WastedEnergy_AC3 :REAL ;
WastedEnergy_AC3_word :WORD ;
WastedEnergy_AC4 :REAL ;
WastedEnergy_AC4_word :WORD ;
WastedEnergy_AC5 :REAL ;
WastedEnergy_AC5_word :WORD ;
WastedEnergy_AC6 :REAL ;
WastedEnergy_AC6_word :WORD ;
Total_PI : REAL ;
// Time variables
Result_time : SysTimeRtc.RTS_IEC_RESULT;
udiLocal_DateAndTime : UDINT;
current_date : UDINT ;

	
END_VAR

IF GVL.startUp THEN
	startupReadcsv();
	IF NOT GVL.startUp THEN	
		GVL.xReadCOP := FALSE;
		GVL.startdelaytimer :=TRUE;
	END_IF
	
END_IF

GVL.delaytimer (IN:= GVL.startdelaytimer, PT:=T#5S);
IF GVL.delaytimer.Q THEN
	GVL.xReadCOP := TRUE;
	GVL.startdelaytimer:=FALSE;
	resetbuttons := TRUE ;
END_IF
delaytimer2 (IN:= resetbuttons, PT:=T#5S);
IF delaytimer2.Q THEN
	GVL.xReadCOP := FALSE;
	GVL.initRead := FALSE;
	resetbuttons := FALSE;
END_IF

// Get system time
current_date := TO_UDINT(SysTimeRtcGet(Result_time));
Result_time := SysTimeRTCConvertUTCToLocal(current_date, udiLocal_DateAndTime);
GVL.CurrentDate := TO_DT(udiLocal_DateAndTime); // DT#2018-6-6-9:8:38

// MWCC
Tot_Q2_MWh:=Tot_Q2:=Chiller_1.Q2_chillerMWh + sequence.Chiller_2_Q2_MWh + Sequence.Chiller_3_Q2_MWh + Sequence.Chiller_4_Q2_MWh + Sequence.Chiller_5_Q2_MWh + Sequence.Chiller_6_Q2_MWh ;
Tot_P1_MWh:=Tot_Q2:=Chiller_1.Chiller_P1_MWh + sequence.Chiller_2_P1_MWh + Sequence.Chiller_3_P1_MWh + Sequence.Chiller_4_P1_MWh + Sequence.Chiller_5_P1_MWh + Sequence.Chiller_6_P1_MWh ;




// New Func
Power_motor_1_kW:=sequence.P1_motor_1_kW;
Power_motor_2_kW:=sequence.P1_motor_2_kW;;
Power_motor_3_kW:=sequence.P1_motor_3_kW;;
(*
Power_motor_4_kW:=Chiller_4.P1_motor_kW;
Power_motor_5_kW:=Chiller_5.P1_motor_kW;
Power_motor_6_kW:=Chiller_6.P1_motor_kW;
*)

Tot_Power_motor:=Power_motor_1_kW + Power_motor_2_kW + Power_motor_3_kW + Power_motor_4_kW;
Tot_Q2:=sequence.Q2kW_chiller_1 + sequence.Q2kW_chiller_2 + Sequence.Q2kW_chiller_3 + Sequence.Q2kW_chiller_4 + Sequence.Q2kW_chiller_5 + Sequence.Q2kW_chiller_6;
// Tot_Q2:=Chiller_1.Chiller_capacity_kW + Chiller_2.Chiller_capacity_kW + Chiller_3.Chiller_capacity_kW + Chiller_4.Chiller_capacity_kW ;
COP_chiller_1:=Chiller_1.COP_chiller_ele;
COP_chiller_2:=Chiller_2.COP_chiller_ele;
COP_chiller_3:=Chiller_3.COP_chiller_ele;
COP_chiller_4:=Chiller_4.COP_chiller_ele;
(*
COP_chiller_5:=Chiller_5.COP_chiller_ele;
COP_chiller_6:=Chiller_6.COP_chiller_ele;
*)
totRunningChillers := BOOL_TO_INT(Chiller_1.Unit_running) + BOOL_TO_INT(Chiller_2.Unit_running) + BOOL_TO_INT(Chiller_3.Unit_running) + BOOL_TO_INT(Chiller_4.Unit_running);

IF Chiller_1.Unit_running THEN
	PI_calculation(Chiller_1.Chiller_capacity,Chiller_1.Temp_water_inlet_cond,COP_chiller_1,Chiller_1.Temp_chilled_medium_out, 1, PI_act=>PI_chiller_1, noCalc_error=>PI_Calc_Error_AC1, COP_theo=>COP_theo_AC1);	
	WastedEnergy_AC1 := Wasted_calc(Chiller_1.Chiller_capacity_kW, COP_theo_AC1, Power_motor_1_kW) ;
	ELSE
	PI_chiller_1 := 0;
	WastedEnergy_AC1 := 0;
	PI_Calc_Error_AC1 := TRUE;
	COP_theo_AC1 := 0;
END_IF

IF Chiller_2.Unit_running THEN
	PI_calculation(Chiller_2.Chiller_capacity,Chiller_2.Temp_water_inlet_cond,COP_chiller_2,Chiller_2.Temp_chilled_medium_out, 1, PI_act=>PI_chiller_2,noCalc_error=>PI_Calc_Error_AC2, COP_theo=>COP_theo_AC2);
	WastedEnergy_AC2 := Wasted_calc(Chiller_2.Chiller_capacity_kW, COP_theo_AC2, Power_motor_2_kW) ;
	ELSE
	PI_chiller_2 := 0;
	WastedEnergy_AC2 := 0;
	PI_Calc_Error_AC2 := TRUE;
	COP_theo_AC2 := 0;
END_IF

IF Chiller_3.Unit_running THEN
	PI_calculation(Chiller_3.Chiller_capacity,Chiller_3.Temp_water_inlet_cond,COP_chiller_3,Chiller_3.Temp_chilled_medium_out, 1, PI_act=>PI_chiller_3,noCalc_error=>PI_Calc_Error_AC3, COP_theo=>COP_theo_AC3);
	WastedEnergy_AC3 := Wasted_calc(Chiller_3.Chiller_capacity_kW, COP_theo_AC3, Power_motor_3_kW) ;
	ELSE
	PI_chiller_3 := 0;
	WastedEnergy_AC3 := 0;	
	PI_Calc_Error_AC3 := TRUE;
	COP_theo_AC3 := 0;
END_IF


(*
IF Chiller_4.Unit_running THEN
	PI_calculation(Chiller_4.Chiller_capacity,Chiller_4.Temp_water_inlet_cond,COP_chiller_4,Chiller_4.Temp_chilled_medium_out, 1, PI_act=>PI_chiller_4,noCalc_error=>PI_Calc_Error_AC4, COP_theo=>COP_theo_AC4);
	WastedEnergy_AC4 := Wasted_calc(Chiller_4.Chiller_capacity_kW, COP_theo_AC4, Power_motor_4_kW) ;
	ELSE
	PI_chiller_4 := 0;
	WastedEnergy_AC4 := 0;
	PI_Calc_Error_AC4 := FALSE;
	COP_theo_AC4 := 0;
END_IF


IF Chiller_5.Unit_running THEN
	PI_calculation(Chiller_5.Chiller_capacity,Chiller_5.Temp_water_inlet_cond,COP_chiller_5,Chiller_5.Temp_chilled_medium_out, 2, PI_act=>PI_chiller_5,noCalc_error=>PI_Calc_Error_AC5, COP_theo=>COP_theo_AC5);
	WastedEnergy_AC5 := Wasted_calc(sequence.Q2kW_chiller_5, COP_theo_AC5, Power_motor_5_kW) ;
	ELSE
	PI_chiller_5 := 0;
	WastedEnergy_AC5 := 0;
	PI_Calc_Error_AC5 := TRUE ;			
END_IF

IF Chiller_6.Unit_running THEN
	PI_calculation(Chiller_6.Chiller_capacity,Chiller_6.Temp_water_inlet_cond,COP_chiller_6,Chiller_6.Temp_chilled_medium_out, 2, PI_act=>PI_chiller_6,noCalc_error=>PI_Calc_Error_AC6, COP_theo=>COP_theo_AC6);
	WastedEnergy_AC6 := Wasted_calc(sequence.Q2kW_chiller_6, COP_theo_AC6, Power_motor_6_kW) ;
	ELSE
	PI_chiller_6 := 0;
	WastedEnergy_AC6 := 0 ;
	PI_Calc_Error_AC6 := TRUE ;			
END_IF
*)


PI_chiller_1_word := REAL_TO_WORD(PI_chiller_1 * 100) ;
PI_chiller_2_word := REAL_TO_WORD(PI_chiller_2 * 100) ;
PI_chiller_3_word := REAL_TO_WORD(PI_chiller_3 * 100) ;
PI_chiller_4_word := REAL_TO_WORD(PI_chiller_4 * 100) ;
PI_chiller_5_word := REAL_TO_WORD(PI_chiller_5 * 100) ;
PI_chiller_6_word := REAL_TO_WORD(PI_chiller_6 * 100) ;

WastedEnergy_AC1_word := REAL_TO_WORD(WastedEnergy_AC1) ;
WastedEnergy_AC2_word := REAL_TO_WORD(WastedEnergy_AC2) ;
WastedEnergy_AC3_word := REAL_TO_WORD(WastedEnergy_AC3) ;
WastedEnergy_AC4_word := REAL_TO_WORD(WastedEnergy_AC4) ;
WastedEnergy_AC5_word := REAL_TO_WORD(WastedEnergy_AC5) ;
WastedEnergy_AC6_word := REAL_TO_WORD(WastedEnergy_AC6) ;



(*
PI_calculation(95,31,4.5,6.1, 1, PI_act=>PI_chiller_1 ,noCalc_error=>PI_Calc_Error_AC1, COP_theo=>COP_theo_AC1);
PI_calculation(92,31,4.5,6.1, 3, PI_act=>PI_chiller_2 ,noCalc_error=>PI_Calc_Error_AC2, COP_theo=>COP_theo_AC2);
PI_calculation(91,31,4.5,6.1, 2, PI_act=>PI_chiller_3 ,noCalc_error=>PI_Calc_Error_AC3, COP_theo=>COP_theo_AC3);
PI_calculation(90,31,4.5,6.1, 3, PI_act=>PI_chiller_4 ,noCalc_error=>PI_Calc_Error_AC4, COP_theo=>COP_theo_AC4);
*)

IF totRunningChillers>0 THEN
	Total_PI:=Tot_PI(PI_chiller_1, PI_chiller_2, PI_chiller_3, PI_chiller_4, PI_chiller_5, PI_chiller_6 , totRunningChillers) ;
	ELSE 
	Total_PI := 0 ;
END_IF

END_PROGRAM

// Device/Application/ConvertDataArray_1
// Helper to convert the data array for the visualization.
FUNCTION_BLOCK ConvertDataArray_1
VAR_INPUT
	xExecute			: BOOL ;
	asData				: ARRAY[0..970] OF STRING(100);
END_VAR
VAR_OUTPUT
	asConvertedCOPData		: ARRAY[0..2, 0..320] OF STRING(100);
	convert_finished 	: BOOL := FALSE ;
END_VAR
VAR
	i				: INT;
	iRow			: INT;
	iColumn			: INT;
END_VAR

IF NOT xExecute THEN
	RETURN;
END_IF
iColumn := 0;
iRow := 0;
FOR i := 0 TO 960 DO
	asConvertedCOPData[iColumn, iRow] := asData[i];
	iColumn := iColumn + 1;
	IF iColumn > 2 THEN
		iColumn := 0;
		iRow := iRow + 1;
	END_IF
END_FOR
convert_finished := TRUE ;

END_FUNCTION_BLOCK

// Device/Application/ConvertDataArray_2
// Helper to convert the data array for the visualization.
FUNCTION_BLOCK ConvertDataArray_2
VAR_INPUT
	xExecute			: BOOL ;
	asData				: ARRAY[0..730] OF STRING(100);
END_VAR
VAR_OUTPUT
	asConvertedData		: ARRAY[0..8, 0..80] OF STRING(100);
	convert_finished 	: BOOL := FALSE ;
END_VAR
VAR
	i				: INT;
	iRow			: INT;
	iColumn			: INT;
END_VAR

IF NOT xExecute THEN
	RETURN;
END_IF
iColumn := 0;
iRow := 0;
FOR i := 0 TO 730 DO
	asConvertedData[iColumn, iRow] := asData[i];
	iColumn := iColumn + 1;
	IF iColumn > 8 THEN
		iColumn := 0;
		iRow := iRow + 1;
	END_IF
END_FOR
convert_finished := TRUE ;

END_FUNCTION_BLOCK

// Device/Application/ConvertDataArray_3
// Helper to convert the data array for the visualization.
FUNCTION_BLOCK ConvertDataArray_3
VAR_INPUT
	xExecute			: BOOL ;
	asData				: ARRAY[0..730] OF STRING(100);
END_VAR
VAR_OUTPUT
	asConvertedData		: ARRAY[0..8, 0..80] OF STRING(100);
	convert_finished 	: BOOL := FALSE ;
END_VAR
VAR
	i				: INT;
	iRow			: INT;
	iColumn			: INT;
END_VAR

IF NOT xExecute THEN
	RETURN;
END_IF
iColumn := 0;
iRow := 0;
FOR i := 0 TO 730 DO
	asConvertedData[iColumn, iRow] := asData[i];
	iColumn := iColumn + 1;
	IF iColumn > 8 THEN
		iColumn := 0;
		iRow := iRow + 1;
	END_IF
END_FOR
convert_finished := TRUE ;

END_FUNCTION_BLOCK

// Device/Application/ConvertDataArray
// Helper to convert the data array for the visualization.
FUNCTION_BLOCK ConvertDataArray
VAR_INPUT
	xExecute			: BOOL ;
	asData				: ARRAY[0..730] OF STRING(100);
END_VAR
VAR_OUTPUT
	asConvertedData		: ARRAY[0..8, 0..80] OF STRING(100);
	convert_finished 	: BOOL := FALSE ;
END_VAR
VAR
	i				: INT;
	iRow			: INT;
	iColumn			: INT;
END_VAR

IF NOT xExecute THEN
	RETURN;
END_IF
iColumn := 0;
iRow := 0;
FOR i := 0 TO 730 DO
	asConvertedData[iColumn, iRow] := asData[i];
	iColumn := iColumn + 1;
	IF iColumn > 8 THEN
		iColumn := 0;
		iRow := iRow + 1;
	END_IF
END_FOR
convert_finished := TRUE ;

END_FUNCTION_BLOCK

// Device/Application/Chiller1Menu
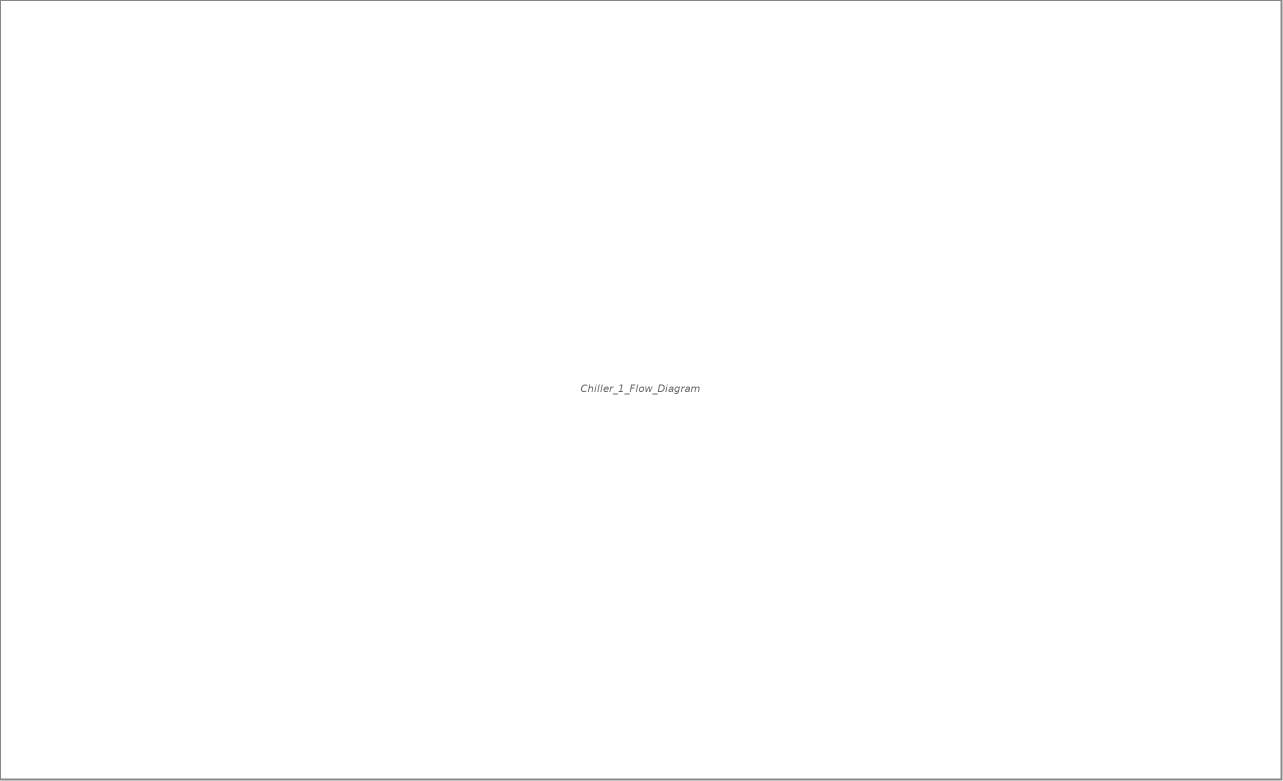
VISUALIZATION Chiller1Menu  // 1283x781
    TabControl (0,-2 1281x781)
        shows Chiller_1_Flow_Diagram()
        shows Chiller_1_Values()
        shows Chiller_1_Alarm()
        shows Chiller_1_Trip()
        shows Chiller_1_Trend()
        shows Chiller_1_Trip()
        [0]: TabTitle=Diagram
        [1]: TabTitle=Measured values
        [2]: TabTitle=Alarm
        [3]: TabTitle=Trip
        [4]: TabTitle=Trend
        [5]: TabTitle=Trip
END_VISUALIZATION

(* text list System (id | default)
  Apr | Apr
  April | April
  Aug | Aug
  August | August
  Dec | Dec
  December | December
  Feb | Feb
  February | February
  Fri | Fri
  Friday | Friday
  Jan | Jan
  January | January
  Jul | Jul
  July | July
  Jun | Jun
  June | June
  Mar | Mar
  March | March
  May | May
  May_3Letter | May
  Mon | Mon
  Monday | Monday
  Nov | Nov
  November | November
  Oct | Oct
  October | October
  Sat | Sat
  Saturday | Saturday
  Sep | Sep
  September | September
  Sun | Sun
  Sunday | Sunday
  Thu | Thu
  Thursday | Thursday
  Tue | Tue
  Tuesday | Tuesday
  Wed | Wed
  Wednesday | Wednesday
   |  *)

(* text list Chiller2Alarmgroup (id | default)
  0 | Chiller_2.T_Overload_compressor_motor
  1 | Chiller_2.T_Starter_failure_trip
  2 | Chiller_2.T_Oil_pump_running_failure
  3 | Chiller_2.T_Overload_oil_pump_motor
  4 | Chiller_2.T_Compressor_running_failure
  5 | Chiller_2.T_Softstarter_failure
  6 | Chiller_2.T_Motorstarter_failure
  7 | Chiller_2.T_Comp_motor_power_loss
  8 | Chiller_2.T_Emergency_stop
  9 | Chiller_2.T_Flow_switch_FT01
  10 | Chiller_2.T_Chilled_pump_run_failure
  11 | Chiller_2.T_CW_valveopen_failure
  12 | Chiller_2.T_Sea_water_pump_run_failure
  13 | Chiller_2.T_SW_valveopen_failure
  14 | Chiller_2.T_Comp_motor_leak_detection
  15 | Chiller_2.T_Cathodic_protec_sys_alarm
  16 | Chiller_2.T_High_discharge_pressure
  17 | Chiller_2.T_Low_discharge_pressure
  18 | Chiller_2.T_Low_suction_pressure
  19 | Chiller_2.T_High_suction_pressure
  20 | Chiller_2.T_High_discharge_temp
  21 | Chiller_2.T_High_temp_oil_inlet_comp
  22 | Chiller_2.T_High_temp_oil_receiver
  23 | Chiller_2.T_Low_temp_oil_receiver
  24 | Chiller_2.T_Low_oil_diff_pressure
  25 | Chiller_2.T_High_diff_oil_pressure
  26 | Chiller_2.T_High_oil_filter_diff_press
  27 | Chiller_2.T_High_disch_superheat
  28 | Chiller_2.T_Low_disch_superheat
  29 | Chiller_2.T_Low_CW_inlet_temp
  30 | Chiller_2.T_High_CW_inlet_temp
  31 | Chiller_2.T_Low_CW_outlet_temp
  32 | Chiller_2.T_High_CW_outlet_temp
  33 | Chiller_2.T_Low_chilled_medium_flow
  34 | Chiller_2.T_High_chilled_medium_flow
  35 | Chiller_2.T_Low_SW_inlet_temp
  36 | Chiller_2.T_High_SW_inlet_temp
  37 | Chiller_2.T_Low_SW_outlet_temp
  38 | Chiller_2.T_High_SW_outlet_temp
  39 | Chiller_2.T_Low_condenser_flow
  40 | Chiller_2.T_High_condenser_flow
  41 | Chiller_2.T_High_motor_wind_temp_R
  42 | Chiller_2.T_High_motor_wind_temp_S
  43 | Chiller_2.T_High_motor_wind_temp_T
  44 | Chiller_2.T_High_comp_motor_DE_bear_temp
  45 | Chiller_2.T_High_comp_motor_NDE_bear_temp
  46 | Chiller_2.T_High_motor_air_temp
  47 | Chiller_2.T_High_comp_motor_DE_bear_vib
  48 | Chiller_2.T_High_comp_motor_NDE_bear_Vib
  49 | Chiller_2.T_High_press_ratio
  50 | Chiller_2.T_Low_press_ratio
  51 | Chiller_2.T_Low_CW_dP
  52 | Chiller_2.T_High_CW_dP
  53 | Chiller_2.T_Low_SW_dP
  54 | Chiller_2.T_High_SW_dP
  55 | Chiller_2.T_Long_time_PRV
  56 | Chiller_2.T_Surge_detection
  57 | Chiller_2.T_Comp_thrust_bearing_position
  58 | Chiller_2.T_Comp_thrust_neg_move
  59 | Chiller_2.T_Comp_thrust_pos_move
  60 | Chiller_2.T_VGD_fault
  61 | Chiller_2.T_Low_liquid_level
  62 | Chiller_2.T_Low_oilpress_prelube
  63 | Chiller_2.T_Low_oilpress_standby
  64 | Chiller_2.T_Sensor_low_signal_AI_64 
  65 | Chiller_2.T_Sensor_high_signal_AI_64 
  66 | Chiller_2.T_Sensor_low_signal_AI_66
  67 | Chiller_2.T_Sensor_high_signal_AI_66 
  68 | Chiller_2.T_Sensor_low_signal_AI_128 
  69 | Chiller_2.T_Sensor_high_signal_AI_128 
  70 | Chiller_2.T_Sensor_low_signal_AI_130 
  71 | Chiller_2.T_Sensor_high_signal_AI_130 
  72 | Chiller_2.T_Sensor_low_signal_AI_132 
  73 | Chiller_2.T_Sensor_high_signal_AI_132 
  74 | Chiller_2.T_Sensor_low_signal_AI_134 
  75 | Chiller_2.T_Sensor_high_signal_AI_134 
  76 | Chiller_2.T_Sensor_low_signal_AI_136 
  77 | Chiller_2.T_Sensor_high_signal_AI_136 
  78 | Chiller_2.T_Sensor_low_signal_AI_138 
  79 | Chiller_2.T_Sensor_high_signal_AI_138 
  80 | Chiller_2.T_Sensor_low_signal_AI_140 
  81 | Chiller_2.T_Sensor_high_signal_AI_140 
  82 | Chiller_2.T_Sensor_low_signal_AI_142 
  83 | Chiller_2.T_Sensor_high_signal_AI_142 
  84 | Chiller_2.T_Sensor_low_signal_AI_144 
  85 | Chiller_2.T_Sensor_high_signal_AI_144 
  86 | Chiller_2.T_Sensor_low_signal_AI_146 
  87 | Chiller_2.T_Sensor_high_signal_AI_146 
  88 | Chiller_2.T_Sensor_low_signal_AI_148 
  89 | Chiller_2.T_Sensor_high_signal_AI_148 
  90 | Chiller_2.T_Sensor_low_signal_AI_150 
  91 | Chiller_2.T_Sensor_high_signal_AI_150 
  92 | Chiller_2.T_Sensor_low_signal_AI_152 
  93 | Chiller_2.T_Sensor_high_signal_AI_152 
  94 | Chiller_2.T_Sensor_low_signal_AI_154 
  95 | Chiller_2.T_Sensor_high_signal_AI_154 
  96 | Chiller_2.T_Sensor_low_signal_AI_156 
  97 | Chiller_2.T_Sensor_high_signal_AI_156 
  98 | Chiller_2.T_Sensor_low_signal_AI_158 
  99 | Chiller_2.T_Sensor_high_signal_AI_158 
  100 | Chiller_2.T_Sensor_low_signal_AI_160 
  101 | Chiller_2.T_Sensor_high_signal_AI_160 
  102 | Chiller_2.T_Sensor_low_signal_AI_162 
  103 | Chiller_2.T_Sensor_high_signal_AI_162 
  104 | Chiller_2.T_Sensor_low_signal_AI_164 
  105 | Chiller_2.T_Sensor_high_signal_AI_164 
  106 | Chiller_2.T_Sensor_low_signal_AI_166 
  107 | Chiller_2.T_Sensor_high_signal_AI_166 
  108 | Chiller_2.T_Sensor_low_signal_AI_168 
  109 | Chiller_2.T_Sensor_high_signal_AI_168 
  110 | Chiller_2.T_Sensor_low_signal_AI_170 
  111 | Chiller_2.T_Sensor_high_signal_AI_170 
  112 | Chiller_2.T_Sensor_low_signal_AI_172 
  113 | Chiller_2.T_Sensor_high_signal_AI_172 
  114 | Chiller_2.T_Sensor_low_signal_AI_174 
  115 | Chiller_2.T_Sensor_high_signal_AI_174 
  116 | Chiller_2.T_Sensor_high_signal_AI_176 
  117 | Chiller_2.T_Sensor_high_signal_AI_178 
  118 | Chiller_2.T_Sensor_high_signal_AI_180 
  119 | Chiller_2.T_Sensor_high_signal_AI_182 
  120 | Chiller_2.T_Sensor_high_signal_AI_184 
  121 | Chiller_2.T_Sensor_high_signal_AI_186 
  122 | Chiller_2.T_Sensor_high_signal_AI_188 
  123 | Chiller_2.T_Sensor_high_signal_AI_190 
  124 | Chiller_2.T_Sensor_high_signal_AI_192 
  125 | Chiller_2.T_Sensor_high_signal_AI_194 
  126 | Chiller_2.T_Sensor_high_signal_AI_196 
  127 | Chiller_2.T_Sensor_high_signal_AI_198 
  128 | Chiller_2.T_Sensor_high_signal_AI_200 
  129 | Chiller_2.T_Sensor_high_signal_AI_202 
  130 | Chiller_2.T_Sensor_high_signal_AI_204 
  131 | Chiller_2.T_Sensor_high_signal_AI_206
  132 | Chiller_2.A_High_control_panel_temp
  133 | Chiller_2.A_high_disch_press
  134 | Chiller_2.A_low_disch_press
  135 | Chiller_2.A_Low_suction_pressure
  136 | Chiller_2.A_High_suction_pressure
  137 | Chiller_2.A_High_discharge_temp 
  138 | Chiller_2.A_High_temp_oil_inlet_comp
  139 | Chiller_2.A_Low_temp_oil_inlet_comp
  140 | Chiller_2.A_High_oil_temp_receiver
  141 | Chiller_2.A_Low_oil_temp_receiver
  142 | Chiller_2.A_Low_oil_diff_pressure
  143 | Chiller_2.A_High_oil_diff_pressure
  144 | Chiller_2.A_Low_discharge_superheat
  145 | Chiller_2.A_High_discharge_superheat
  146 | Chiller_2.A_Low_CW_inlet_temp
  147 | Chiller_2.A_High_CW_inlet_temp
  148 | Chiller_2.A_Low_CW_outlet_temp
  149 | Chiller_2.A_High_CW_outlet_temp
  150 | Chiller_2.A_Low_chilled_medium_flow
  151 | Chiller_2.A_High_chilled_medium_flow
  152 | Chiller_2.A_Low_condenser_flow
  153 | Chiller_2.A_High_condenser_flow
  154 | Chiller_2.A_High_press_ratio
  155 | Chiller_2.A_Low_press_ratio
  156 | Chiller_2.A_Motor_speed_low 
  157 | Chiller_2.A_Low_SW_inlet_temp 
  158 | Chiller_2.A_High_SW_inlet_temp 
  159 | Chiller_2.A_Low_SW_outlet_temp 
  160 | Chiller_2.A_High_SW_outlet_temp
  161 | Chiller_2.A_High_suction_superheat
  162 | Chiller_2.A_Low_suction_superheat
  163 | Chiller_2.A_High_oil_filter_diff_press
  164 | Chiller_2.A_High_CW_dP
  165 | Chiller_2.A_Low_CW_dP
  166 | Chiller_2.A_High_temp_oil_separator
  167 | Chiller_2.A_Low_temp_oil_separator
  168 | Chiller_2.A_High_motor_wind_temp_R
  169 | Chiller_2.A_High_motor_wind_temp_S
  170 | Chiller_2.A_High_motor_wind_temp_T
  171 | Chiller_2.A_High_comp_mo_DE_bear_temp
  172 | Chiller_2.A_High_comp_mo_NDE_bear_temp
  173 | Chiller_2.A_High_motor_air_temp
  174 | Chiller_2.A_High_comp_mo_DE_bear_vib
  175 | Chiller_2.A_High_comp_mo_NDE_bear_vib
  176 | Chiller_2.A_High_CW_dP  
  177 | Chiller_2.A_Low_CW_dP 
  178 | Chiller_2.A_High_SW_dP 
  179 | Chiller_2.A_Low_SW_dP
  180 | Chiller_2.A_VGD_Fault
  181 | Chiller_2.A_Low_liquid_level
   |  *)

(* text list Chiller_trendvalues (id | default)
  0 | Clear values
  17 | Temp Chilled Medium In
  18 | Temp Chilled Medium Out
  1 | Chiller Capacity
  5 | Setpoint Liquid Level
  7 | Feedback PRV
  9 | Feedback VGD
  8 | Feedback Sea Water Valve Overboard
  6 | Feedback Liquid Valve
  11 | Liquid Level Condenser
  13 | Motor Current
  19 | Temp Discharge Gas
  22 | Temp Motor Air
  23 | Temp Motor Bearing DE
  24 | Temp Motor Bearing NDE
  25 | Temp Motor Winding R
  26 | Temp Motor Winding S
  27 | Temp Motor Winding T
  31 | Temp Trafo Wind U
  3 | dP CW
  20 | Temp Discharge Saturated
  15 | Order VFD Hz
  35 | Thrust Bearing position
  34 | Theta Out
  21 | Temp Discharge Superheat
  4 | dP SW
  28 | Temp Oil Inlet Compressor
  33 | Temp Trafo wind W
  12 | Liquid Valve Output
  10 | Hot Gas Valve Output
  16 | Speed Feedback VFD
  29 | Temp Sea Water Inlet
  14 | Oil Diff Pressure
  2 | Control Signal SW Valve
  32 | Temp Trafo Wind V
  30 | Temp Suction Saturated
   |  *)
